C07278=1088.275,-115.195,449.756,174.378,16.605,152.666
C07279=1088.269,-115.445,449.766,174.377,16.605,152.667
C07280=1088.263,-115.695,449.776,174.375,16.604,152.667
C07281=1088.257,-115.945,449.785,174.373,16.603,152.667
C07282=1088.251,-116.194,449.795,174.372,16.603,152.667
C07283=1088.245,-116.444,449.804,174.370,16.603,152.667
C07284=1088.239,-116.693,449.813,174.369,16.602,152.668
C07285=1088.233,-116.943,449.823,174.368,16.602,152.668
C07286=1088.227,-117.193,449.833,174.366,16.601,152.668
C07287=1088.220,-117.443,449.842,174.364,16.600,152.668
C07288=1088.215,-117.693,449.851,174.363,16.600,152.668
C07289=1088.208,-117.943,449.861,174.361,16.599,152.669
C07290=1088.202,-118.193,449.870,174.359,16.598,152.669
C07291=1088.197,-118.442,449.879,174.358,16.598,152.669
C07292=1088.190,-118.691,449.888,174.356,16.597,152.669
C07293=1088.184,-118.941,449.898,174.355,16.596,152.669
C07294=1088.177,-119.191,449.907,174.354,16.596,152.670
C07295=1088.171,-119.441,449.917,174.352,16.596,152.670
C07296=1088.165,-119.691,449.927,174.350,16.595,152.670
C07297=1088.159,-119.941,449.935,174.348,16.594,152.670
C07298=1088.153,-120.191,449.945,174.347,16.594,152.670
C07299=1088.147,-120.440,449.954,174.345,16.593,152.671
C07300=1088.141,-120.689,449.963,174.343,16.592,152.671
C07301=1088.134,-120.939,449.973,174.342,16.592,152.671
C07302=1088.128,-121.189,449.982,174.340,16.592,152.671
C07303=1088.122,-121.439,449.991,174.340,16.591,152.671
C07304=1088.116,-121.689,450.001,174.338,16.590,152.672
C07305=1088.110,-121.939,450.010,174.336,16.590,152.672
C07306=1088.104,-122.188,450.019,174.335,16.590,152.672
C07307=1088.098,-122.438,450.028,174.333,16.589,152.672
C07308=1088.091,-122.687,450.038,174.331,16.588,152.673
C07309=1088.086,-122.938,450.047,174.330,16.588,152.673
C07310=1088.079,-123.188,450.056,174.328,16.587,152.673
C07311=1088.074,-123.437,450.066,174.326,16.586,152.673
C07312=1088.068,-123.686,450.075,174.325,16.586,152.673
C07313=1088.061,-123.937,450.083,174.323,16.586,152.674
C07314=1088.055,-124.186,450.093,174.322,16.585,152.674
C07315=1088.049,-124.436,450.103,174.321,16.585,152.674
C07316=1088.042,-124.686,450.112,174.319,16.584,152.674
C07317=1088.037,-124.936,450.121,174.317,16.583,152.674
C07318=1088.030,-125.185,450.130,174.316,16.583,152.675
C07319=1088.024,-125.435,450.139,174.314,16.583,152.675
C07320=1088.018,-125.685,450.149,174.312,16.582,152.675
C07321=1088.012,-125.935,450.158,174.311,16.582,152.675
C07322=1088.006,-126.184,450.166,174.309,16.581,152.676
C07323=1088.000,-126.434,450.176,174.308,16.581,152.676
C07324=1087.993,-126.684,450.185,174.306,16.580,152.676
C07325=1087.987,-126.934,450.194,174.304,16.580,152.676
C07326=1087.981,-127.183,450.203,174.303,16.580,152.677
C07327=1087.974,-127.433,450.213,174.302,16.579,152.677
C07328=1087.969,-127.683,450.221,174.300,16.578,152.677
C07329=1087.962,-127.941,450.231,174.299,16.578,152.677
C07330=1087.957,-128.198,450.240,174.297,16.577,152.677
C07331=1087.958,-128.455,450.252,174.296,16.575,152.677
C07332=1087.965,-128.710,450.265,174.296,16.571,152.676
C07333=1087.560,-128.731,450.140,174.254,16.677,152.705
C07334=1087.553,-128.477,450.127,174.254,16.681,152.706
C07335=1087.552,-128.220,450.115,174.255,16.683,152.706
C07336=1087.558,-127.963,450.105,174.257,16.684,152.706
C07337=1087.564,-127.705,450.096,174.258,16.684,152.705
C07338=1087.571,-127.455,450.086,174.260,16.685,152.705
C07339=1087.576,-127.205,450.078,174.262,16.686,152.705
C07340=1087.582,-126.955,450.068,174.263,16.686,152.705
C07341=1087.589,-126.706,450.059,174.265,16.687,152.705
C07342=1087.595,-126.456,450.050,174.267,16.687,152.704
C07343=1087.601,-126.206,450.041,174.268,16.687,152.704
C07344=1087.607,-125.957,450.031,174.270,16.688,152.704
C07345=1087.614,-125.707,450.022,174.271,16.689,152.704
C07346=1087.619,-125.457,450.014,174.272,16.689,152.703
C07347=1087.626,-125.207,450.004,174.274,16.690,152.703
C07348=1087.632,-124.957,449.995,174.275,16.690,152.703
C07349=1087.639,-124.708,449.986,174.277,16.691,152.703
C07350=1087.644,-124.458,449.977,174.279,16.691,152.703
C07351=1087.650,-124.208,449.967,174.280,16.691,152.702
C07352=1087.656,-123.958,449.958,174.282,16.692,152.702
C07353=1087.663,-123.709,449.949,174.284,16.693,152.702
C07354=1087.669,-123.458,449.940,174.285,16.693,152.702
C07355=1087.675,-123.209,449.931,174.287,16.694,152.701
C07356=1087.681,-122.960,449.921,174.289,16.694,152.701
C07357=1087.687,-122.710,449.912,174.289,16.695,152.701
C07358=1087.693,-122.460,449.902,174.291,16.696,152.701
C07359=1087.700,-122.210,449.894,174.293,16.696,152.701
C07360=1087.706,-121.960,449.884,174.294,16.697,152.701
C07361=1087.711,-121.711,449.875,174.296,16.697,152.700
C07362=1087.718,-121.461,449.866,174.298,16.698,152.700
C07363=1087.724,-121.211,449.856,174.299,16.698,152.700
C07364=1087.730,-120.961,449.847,174.301,16.699,152.700
C07365=1087.736,-120.711,449.838,174.303,16.700,152.699
C07366=1087.743,-120.462,449.829,174.304,16.700,152.699
C07367=1087.748,-120.213,449.819,174.305,16.701,152.699
C07368=1087.754,-119.963,449.810,174.307,16.701,152.699
C07369=1087.761,-119.713,449.800,174.308,16.701,152.699
C07370=1087.767,-119.463,449.791,174.310,16.702,152.698
C07371=1087.773,-119.213,449.782,174.312,16.703,152.698
C07372=1087.779,-118.963,449.772,174.313,16.703,152.698
C07373=1087.785,-118.713,449.763,174.315,16.704,152.698
C07374=1087.792,-118.464,449.754,174.316,16.705,152.698
C07375=1087.798,-118.215,449.745,174.318,16.705,152.697
C07376=1087.804,-117.965,449.735,174.319,16.706,152.697
C07377=1087.810,-117.715,449.725,174.321,16.706,152.697
C07378=1087.816,-117.465,449.716,174.323,16.708,152.697
C07379=1087.822,-117.215,449.706,174.324,16.708,152.697
C07380=1087.828,-116.966,449.697,174.326,16.708,152.696
C07381=1087.835,-116.716,449.687,174.327,16.709,152.696
C07382=1087.840,-116.465,449.678,174.329,16.709,152.696
C07383=1087.847,-116.216,449.669,174.330,16.710,152.696
C07384=1087.852,-115.967,449.660,174.332,16.711,152.696
C07385=1087.858,-115.717,449.650,174.333,16.711,152.696
C07386=1087.864,-115.467,449.640,174.335,16.712,152.695
C07387=1087.871,-115.217,449.631,174.337,16.713,152.695
C07388=1087.877,-114.967,449.621,174.338,16.714,152.695
C07389=1087.883,-114.718,449.612,174.339,16.714,152.695
C07390=1087.889,-114.468,449.602,174.341,16.714,152.695
C07391=1087.895,-114.218,449.593,174.343,16.716,152.694
C07392=1087.902,-113.968,449.583,174.344,16.716,152.694
C07393=1087.908,-113.718,449.573,174.346,16.717,152.694
C07394=1087.915,-113.448,449.563,174.348,16.717,152.694
C07395=1087.921,-113.177,449.553,174.349,16.718,152.694
C07396=1087.928,-112.907,449.542,174.351,16.719,152.693
C07397=1087.934,-112.635,449.532,174.353,16.720,152.693
C07398=1087.940,-112.385,449.523,174.354,16.720,152.693
C07399=1087.947,-112.135,449.513,174.356,16.721,152.693
C07400=1087.953,-111.886,449.503,174.358,16.722,152.693
C07401=1087.959,-111.636,449.494,174.359,16.722,152.693
C07402=1087.964,-111.387,449.485,174.360,16.723,152.692
C07403=1087.971,-111.137,449.475,174.362,16.724,152.692
C07404=1087.977,-110.887,449.466,174.364,16.725,152.692
C07405=1087.983,-110.638,449.455,174.365,16.725,152.692
C07406=1087.989,-110.388,449.446,174.367,16.726,152.692
C07407=1087.995,-110.138,449.436,174.368,16.726,152.691
C07408=1088.001,-109.888,449.426,174.369,16.727,152.691
C07409=1088.007,-109.639,449.416,174.371,16.728,152.691
C07410=1088.013,-109.389,449.407,174.373,16.729,152.691
C07411=1088.020,-109.139,449.397,174.375,16.729,152.691
C07412=1088.026,-108.889,449.388,174.376,16.730,152.691
C07413=1088.032,-108.639,449.378,174.377,16.730,152.690
C07414=1088.038,-108.390,449.369,174.379,16.731,152.690
C07415=1088.045,-108.140,449.358,174.381,16.732,152.690
C07416=1088.051,-107.891,449.349,174.382,16.733,152.690
C07417=1088.057,-107.641,449.339,174.383,16.734,152.690
C07418=1088.062,-107.391,449.329,174.385,16.734,152.690
C07419=1088.068,-107.141,449.319,174.387,16.735,152.689
C07420=1088.075,-106.891,449.310,174.388,16.735,152.689
C07421=1088.081,-106.642,449.300,174.390,16.737,152.689
C07422=1088.087,-106.392,449.290,174.392,16.737,152.689
C07423=1088.093,-106.142,449.280,174.393,16.738,152.689
C07424=1088.099,-105.892,449.270,174.394,16.739,152.689
C07425=1088.105,-105.642,449.261,174.396,16.739,152.688
C07426=1088.111,-105.393,449.251,174.398,16.740,152.688
C07427=1088.118,-105.143,449.241,174.400,16.741,152.688
C07428=1088.123,-104.893,449.231,174.400,16.742,152.688
C07429=1088.129,-104.643,449.221,174.402,16.743,152.688
C07430=1088.136,-104.394,449.212,174.404,16.743,152.688
C07431=1088.142,-104.145,449.201,174.406,16.744,152.687
C07432=1088.147,-103.894,449.191,174.407,16.746,152.687
C07433=1088.154,-103.645,449.182,174.408,16.746,152.687
C07434=1088.160,-103.395,449.172,174.410,16.747,152.687
C07435=1088.166,-103.145,449.162,174.412,16.747,152.687
C07436=1088.172,-102.896,449.152,174.413,16.748,152.687
C07437=1088.178,-102.646,449.142,174.414,16.749,152.687
C07438=1088.184,-102.396,449.132,174.416,16.750,152.686
C07439=1088.190,-102.147,449.122,174.418,16.751,152.686
C07440=1088.196,-101.897,449.112,174.419,16.752,152.686
C07441=1088.202,-101.647,449.102,174.421,16.752,152.686
C07442=1088.208,-101.397,449.093,174.422,16.753,152.686
C07443=1088.215,-101.148,449.083,174.424,16.754,152.686
C07444=1088.220,-100.898,449.072,174.426,16.755,152.685
C07445=1088.226,-100.648,449.063,174.427,16.756,152.685
C07446=1088.233,-100.399,449.053,174.428,16.756,152.685
C07447=1088.238,-100.149,449.042,174.430,16.757,152.685
C07448=1088.244,-99.899,449.033,174.432,16.758,152.685
C07449=1088.251,-99.650,449.023,174.433,16.759,152.685
C07450=1088.257,-99.400,449.013,174.435,16.760,152.684
C07451=1088.263,-99.150,449.003,174.436,16.760,152.684
C07452=1088.269,-98.901,448.992,174.438,16.761,152.684
C07453=1088.275,-98.651,448.983,174.440,16.762,152.684
C07454=1088.281,-98.401,448.973,174.441,16.763,152.684
C07455=1088.288,-98.151,448.962,174.443,16.764,152.684
C07456=1088.294,-97.901,448.953,174.444,16.765,152.684
C07457=1088.300,-97.652,448.942,174.446,16.765,152.684
C07458=1088.306,-97.375,448.931,174.447,16.766,152.683
C07459=1088.312,-97.099,448.920,174.449,16.767,152.683
C07460=1088.319,-96.822,448.909,174.451,16.769,152.683
C07461=1088.326,-96.546,448.897,174.452,16.769,152.683
C07462=1088.331,-96.296,448.887,174.454,16.770,152.683
C07463=1088.338,-96.047,448.877,174.456,16.771,152.683
C07464=1088.343,-95.796,448.867,174.457,16.772,152.683
C07465=1088.349,-95.547,448.857,174.458,16.773,152.683
C07466=1088.356,-95.296,448.846,174.460,16.774,152.682
C07467=1088.362,-95.047,448.836,174.462,16.775,152.682
C07468=1088.368,-94.797,448.826,174.463,16.776,152.682
C07469=1088.374,-94.547,448.816,174.465,16.777,152.682
C07470=1088.380,-94.298,448.806,174.467,16.778,152.682
C07471=1088.386,-94.048,448.795,174.468,16.778,152.682
C07472=1088.392,-93.799,448.785,174.469,16.779,152.681
C07473=1088.398,-93.549,448.775,174.471,16.780,152.681
C07474=1088.403,-93.299,448.765,174.473,16.781,152.681
C07475=1088.410,-93.050,448.755,174.474,16.782,152.681
C07476=1088.415,-92.799,448.744,174.476,16.784,152.681
C07477=1088.422,-92.550,448.734,174.477,16.784,152.681
C07478=1088.427,-92.300,448.724,174.479,16.785,152.681
C07479=1088.434,-92.050,448.713,174.480,16.786,152.681
C07480=1088.440,-91.801,448.702,174.482,16.787,152.680
C07481=1088.446,-91.551,448.693,174.484,16.788,152.680
C07482=1088.452,-91.301,448.682,174.485,16.789,152.680
C07483=1088.458,-91.052,448.672,174.486,16.789,152.680
C07484=1088.464,-90.802,448.662,174.488,16.790,152.680
C07485=1088.470,-90.552,448.652,174.490,16.791,152.680
C07486=1088.475,-90.303,448.641,174.491,16.792,152.680
C07487=1088.482,-90.053,448.632,174.493,16.794,152.680
C07488=1088.488,-89.803,448.620,174.494,16.795,152.679
C07489=1088.494,-89.553,448.609,174.495,16.795,152.679
C07490=1088.500,-89.304,448.600,174.497,16.796,152.679
C07491=1088.506,-89.054,448.589,174.499,16.797,152.679
C07492=1088.512,-88.804,448.579,174.500,16.798,152.679
C07493=1088.518,-88.555,448.569,174.502,16.799,152.679
C07494=1088.524,-88.306,448.558,174.504,16.800,152.679
C07495=1088.530,-88.055,448.548,174.505,16.801,152.679
C07496=1088.537,-87.806,448.537,174.506,16.802,152.679
C07497=1088.542,-87.556,448.527,174.508,16.803,152.678
C07498=1088.548,-87.306,448.516,174.509,16.804,152.678
C07499=1088.554,-87.057,448.506,174.511,16.805,152.678
C07500=1088.560,-86.806,448.496,174.513,16.806,152.678
C07501=1088.567,-86.557,448.485,174.515,16.807,152.678
C07502=1088.572,-86.307,448.474,174.516,16.808,152.678
C07503=1088.578,-86.057,448.464,174.517,16.809,152.678
C07504=1088.584,-85.808,448.454,174.519,16.810,152.678
C07505=1088.590,-85.559,448.443,174.520,16.811,152.677
C07506=1088.597,-85.308,448.433,174.522,16.812,152.677
C07507=1088.603,-85.059,448.422,174.524,16.813,152.677
C07508=1088.608,-84.809,448.411,174.525,16.814,152.677
C07509=1088.615,-84.560,448.401,174.527,16.815,152.677
C07510=1088.621,-84.309,448.391,174.529,16.816,152.677
C07511=1088.627,-84.060,448.380,174.530,16.816,152.677
C07512=1088.633,-83.810,448.369,174.531,16.817,152.677
C07513=1088.639,-83.560,448.359,174.533,16.819,152.676
C07514=1088.645,-83.311,448.349,174.534,16.820,152.676
C07515=1088.651,-83.061,448.338,174.536,16.821,152.676
C07516=1088.657,-82.812,448.327,174.538,16.822,152.676
C07517=1088.663,-82.562,448.317,174.539,16.823,152.676
C07518=1088.669,-82.312,448.306,174.541,16.824,152.676
C07519=1088.676,-82.062,448.296,174.542,16.825,152.676
C07520=1088.682,-81.813,448.285,174.543,16.826,152.676
C07521=1088.688,-81.563,448.274,174.545,16.827,152.676
C07522=1088.695,-81.289,448.263,174.547,16.828,152.676
C07523=1088.701,-81.015,448.251,174.548,16.829,152.675
C07524=1088.707,-80.740,448.239,174.551,16.831,152.675
C07525=1088.715,-80.466,448.228,174.553,16.831,152.675
C07526=1088.721,-80.216,448.217,174.553,16.832,152.675
C07527=1088.727,-79.966,448.207,174.555,16.833,152.675
C07528=1088.733,-79.717,448.196,174.557,16.834,152.675
C07529=1088.739,-79.467,448.185,174.558,16.835,152.675
C07530=1088.745,-79.217,448.174,174.560,16.836,152.675
C07531=1088.751,-78.968,448.163,174.561,16.838,152.675
C07532=1088.756,-78.718,448.152,174.563,16.839,152.674
C07533=1088.763,-78.468,448.143,174.565,16.840,152.674
C07534=1088.769,-78.218,448.131,174.566,16.841,152.674
C07535=1088.775,-77.969,448.121,174.568,16.842,152.674
C07536=1088.780,-77.719,448.110,174.570,16.843,152.674
C07537=1088.786,-77.470,448.099,174.570,16.844,152.674
C07538=1088.793,-77.220,448.088,174.572,16.845,152.674
C07539=1088.799,-76.970,448.077,174.574,16.846,152.674
C07540=1088.805,-76.721,448.066,174.575,16.847,152.674
C07541=1088.810,-76.471,448.055,174.577,16.848,152.674
C07542=1088.816,-76.220,448.045,174.578,16.850,152.673
C07543=1088.822,-75.971,448.034,174.580,16.851,152.673
C07544=1088.828,-75.722,448.023,174.582,16.852,152.673
C07545=1088.835,-75.472,448.013,174.583,16.853,152.673
C07546=1088.841,-75.222,448.002,174.585,16.854,152.673
C07547=1088.846,-74.973,447.991,174.587,16.855,152.673
C07548=1088.852,-74.723,447.980,174.588,16.856,152.673
C07549=1088.859,-74.473,447.969,174.590,16.858,152.673
C07550=1088.864,-74.223,447.958,174.591,16.859,152.673
C07551=1088.870,-73.974,447.947,174.592,16.859,152.673
C07552=1088.876,-73.724,447.936,174.594,16.861,152.673
C07553=1088.882,-73.474,447.925,174.595,16.862,152.672
C07554=1088.888,-73.225,447.914,174.597,16.863,152.672
C07555=1088.894,-72.975,447.903,174.599,16.864,152.672
C07556=1088.900,-72.725,447.892,174.600,16.865,152.672
C07557=1088.906,-72.476,447.881,174.602,16.867,152.672
C07558=1088.911,-72.226,447.870,174.603,16.868,152.672
C07559=1088.917,-71.977,447.859,174.605,16.869,152.672
C07560=1088.923,-71.726,447.848,174.606,16.870,152.672
C07561=1088.929,-71.477,447.837,174.608,16.871,152.672
C07562=1088.935,-71.228,447.826,174.609,16.873,152.672
C07563=1088.941,-70.978,447.815,174.611,16.874,152.672
C07564=1088.947,-70.728,447.804,174.613,16.875,152.672
C07565=1088.953,-70.478,447.793,174.614,16.876,152.671
C07566=1088.958,-70.229,447.782,174.616,16.877,152.671
C07567=1088.964,-69.978,447.770,174.617,16.879,152.671
C07568=1088.970,-69.729,447.760,174.619,16.880,152.671
C07569=1088.976,-69.479,447.749,174.621,16.881,152.671
C07570=1088.982,-69.230,447.737,174.622,16.882,152.671
C07571=1088.988,-68.980,447.726,174.623,16.883,152.671
C07572=1088.994,-68.731,447.715,174.624,16.884,152.671
C07573=1088.999,-68.481,447.704,174.626,16.885,152.671
C07574=1089.006,-68.231,447.693,174.628,16.886,152.671
C07575=1089.012,-67.982,447.682,174.629,16.887,152.671
C07576=1089.017,-67.732,447.671,174.631,16.889,152.671
C07577=1089.023,-67.482,447.659,174.632,16.890,152.671
C07578=1089.029,-67.232,447.648,174.634,16.891,152.671
C07579=1089.035,-66.983,447.636,174.636,16.892,152.670
C07580=1089.041,-66.733,447.626,174.637,16.893,152.670
C07581=1089.047,-66.484,447.615,174.639,16.895,152.670
C07582=1089.053,-66.233,447.603,174.640,16.896,152.670
C07583=1089.059,-65.984,447.593,174.642,16.897,152.670
C07584=1089.065,-65.734,447.582,174.643,16.898,152.670
C07585=1089.071,-65.485,447.570,174.645,16.900,152.670
C07586=1089.077,-65.213,447.557,174.646,16.901,152.670
C07587=1089.084,-64.941,447.545,174.648,16.902,152.670
C07588=1089.090,-64.668,447.533,174.650,16.904,152.670
C07589=1089.097,-64.396,447.521,174.652,16.905,152.670
C07590=1089.102,-64.147,447.510,174.654,16.906,152.669
C07591=1089.109,-63.897,447.499,174.655,16.908,152.670
C07592=1089.114,-63.647,447.487,174.657,16.909,152.669
C07593=1089.120,-63.398,447.475,174.658,16.910,152.669
C07594=1089.126,-63.148,447.464,174.660,16.911,152.669
C07595=1089.132,-62.898,447.453,174.661,16.913,152.669
C07596=1089.138,-62.648,447.442,174.663,16.914,152.669
C07597=1089.144,-62.399,447.430,174.665,16.915,152.669
C07598=1089.150,-62.149,447.419,174.666,16.916,152.669
C07599=1089.156,-61.899,447.408,174.668,16.918,152.669
C07600=1089.162,-61.650,447.396,174.669,16.919,152.669
C07601=1089.168,-61.400,447.385,174.671,16.920,152.669
C07602=1089.174,-61.151,447.374,174.672,16.921,152.669
C07603=1089.180,-60.901,447.362,174.674,16.922,152.669
C07604=1089.185,-60.651,447.351,174.675,16.924,152.669
C07605=1089.192,-60.401,447.339,174.677,16.925,152.668
C07606=1089.198,-60.152,447.328,174.679,16.926,152.668
C07607=1089.204,-59.902,447.317,174.680,16.927,152.668
C07608=1089.210,-59.653,447.306,174.682,16.929,152.668
C07609=1089.215,-59.403,447.293,174.683,16.930,152.668
C07610=1089.222,-59.153,447.282,174.685,16.931,152.668
C07611=1089.227,-58.904,447.271,174.686,16.932,152.668
C07612=1089.234,-58.654,447.259,174.688,16.933,152.668
C07613=1089.239,-58.404,447.248,174.690,16.935,152.668
C07614=1089.245,-58.154,447.237,174.691,16.936,152.668
C07615=1089.251,-57.905,447.225,174.693,16.937,152.668
C07616=1089.258,-57.655,447.214,174.694,16.938,152.668
C07617=1089.264,-57.406,447.202,174.696,16.939,152.668
C07618=1089.269,-57.156,447.190,174.697,16.941,152.668
C07619=1089.275,-56.907,447.179,174.699,16.942,152.668
C07620=1089.282,-56.657,447.168,174.700,16.943,152.667
C07621=1089.287,-56.407,447.157,174.702,16.944,152.667
C07622=1089.293,-56.157,447.144,174.704,16.946,152.667
C07623=1089.300,-55.907,447.133,174.705,16.947,152.667
C07624=1089.306,-55.658,447.121,174.707,16.948,152.667
C07625=1089.312,-55.408,447.110,174.708,16.949,152.667
C07626=1089.317,-55.159,447.098,174.710,16.951,152.667
C07627=1089.324,-54.909,447.087,174.711,16.952,152.667
C07628=1089.330,-54.660,447.075,174.713,16.953,152.667
C07629=1089.336,-54.410,447.064,174.715,16.954,152.667
C07630=1089.341,-54.161,447.052,174.716,16.956,152.667
C07631=1089.348,-53.910,447.040,174.718,16.957,152.667
C07632=1089.354,-53.661,447.028,174.719,16.958,152.667
C07633=1089.360,-53.411,447.018,174.721,16.959,152.667
C07634=1089.366,-53.161,447.005,174.722,16.961,152.667
C07635=1089.372,-52.912,446.994,174.724,16.962,152.666
C07636=1089.378,-52.662,446.982,174.725,16.963,152.666
C07637=1089.383,-52.412,446.971,174.727,16.965,152.666
C07638=1089.390,-52.163,446.959,174.728,16.966,152.666
C07639=1089.396,-51.913,446.947,174.730,16.967,152.666
C07640=1089.402,-51.664,446.935,174.732,16.968,152.666
C07641=1089.408,-51.414,446.923,174.734,16.970,152.666
C07642=1089.414,-51.164,446.912,174.735,16.971,152.666
C07643=1089.421,-50.915,446.900,174.737,16.972,152.666
C07644=1089.426,-50.664,446.889,174.738,16.974,152.666
C07645=1089.432,-50.416,446.877,174.740,16.975,152.666
C07646=1089.438,-50.166,446.865,174.742,16.976,152.666
C07647=1089.444,-49.916,446.854,174.743,16.978,152.666
C07648=1089.450,-49.666,446.841,174.745,16.979,152.666
C07649=1089.456,-49.417,446.830,174.746,16.980,152.666
C07650=1089.462,-49.146,446.816,174.748,16.982,152.666
C07651=1089.469,-48.875,446.804,174.749,16.983,152.666
C07652=1089.474,-48.604,446.791,174.751,16.985,152.666
C07653=1089.481,-48.334,446.779,174.753,16.986,152.665
C07654=1089.487,-48.084,446.766,174.754,16.988,152.665
C07655=1089.494,-47.834,446.754,174.756,16.989,152.665
C07656=1089.499,-47.584,446.743,174.758,16.990,152.665
C07657=1089.505,-47.335,446.731,174.759,16.991,152.665
C07658=1089.510,-47.086,446.718,174.761,16.992,152.665
C07659=1089.517,-46.835,446.707,174.762,16.994,152.665
C07660=1089.522,-46.586,446.695,174.764,16.995,152.665
C07661=1089.529,-46.337,446.683,174.765,16.996,152.665
C07662=1089.534,-46.086,446.671,174.768,16.998,152.665
C07663=1089.540,-45.837,446.659,174.769,17.000,152.665
C07664=1089.546,-45.587,446.647,174.770,17.001,152.665
C07665=1089.552,-45.338,446.635,174.772,17.002,152.665
C07666=1089.558,-45.088,446.624,174.774,17.003,152.665
C07667=1089.564,-44.838,446.611,174.775,17.005,152.665
C07668=1089.569,-44.589,446.599,174.777,17.006,152.665
C07669=1089.576,-44.339,446.587,174.778,17.008,152.665
C07670=1089.581,-44.089,446.575,174.780,17.009,152.665
C07671=1089.587,-43.840,446.564,174.781,17.010,152.665
C07672=1089.593,-43.590,446.551,174.783,17.012,152.665
C07673=1089.599,-43.341,446.539,174.784,17.013,152.664
C07674=1089.605,-43.091,446.527,174.786,17.014,152.665
C07675=1089.611,-42.841,446.515,174.788,17.016,152.664
C07676=1089.617,-42.592,446.503,174.789,17.018,152.664
C07677=1089.623,-42.342,446.491,174.791,17.019,152.664
C07678=1089.629,-42.092,446.478,174.793,17.020,152.664
C07679=1089.635,-41.843,446.467,174.794,17.021,152.664
C07680=1089.640,-41.593,446.455,174.796,17.022,152.664
C07681=1089.646,-41.343,446.442,174.797,17.024,152.664
C07682=1089.652,-41.094,446.431,174.799,17.025,152.664
C07683=1089.658,-40.844,446.418,174.800,17.026,152.664
C07684=1089.665,-40.595,446.406,174.802,17.028,152.664
C07685=1089.670,-40.345,446.394,174.803,17.029,152.664
C07686=1089.676,-40.096,446.381,174.806,17.031,152.664
C07687=1089.683,-39.845,446.370,174.807,17.032,152.664
C07688=1089.688,-39.596,446.358,174.809,17.034,152.664
C07689=1089.694,-39.346,446.345,174.810,17.035,152.664
C07690=1089.700,-39.097,446.334,174.812,17.036,152.664
C07691=1089.706,-38.847,446.321,174.813,17.038,152.664
C07692=1089.712,-38.598,446.309,174.815,17.039,152.664
C07693=1089.717,-38.348,446.296,174.816,17.040,152.664
C07694=1089.724,-38.098,446.284,174.818,17.042,152.664
C07695=1089.729,-37.849,446.272,174.820,17.044,152.664
C07696=1089.735,-37.599,446.260,174.822,17.045,152.663
C07697=1089.741,-37.349,446.247,174.823,17.046,152.663
C07698=1089.747,-37.100,446.235,174.825,17.048,152.663
C07699=1089.753,-36.851,446.223,174.826,17.049,152.663
C07700=1089.759,-36.601,446.210,174.828,17.050,152.663
C07701=1089.764,-36.351,446.198,174.829,17.052,152.663
C07702=1089.770,-36.102,446.186,174.831,17.053,152.663
C07703=1089.776,-35.852,446.173,174.832,17.055,152.663
C07704=1089.781,-35.602,446.162,174.834,17.056,152.663
C07705=1089.788,-35.352,446.150,174.836,17.058,152.663
C07706=1089.794,-35.103,446.136,174.837,17.059,152.663
C07707=1089.800,-34.853,446.124,174.839,17.061,152.663
C07708=1089.805,-34.604,446.112,174.840,17.062,152.663
C07709=1089.811,-34.354,446.099,174.842,17.063,152.663
C07710=1089.817,-34.104,446.086,174.843,17.064,152.663
C07711=1089.823,-33.854,446.074,174.845,17.066,152.663
C07712=1089.829,-33.606,446.062,174.847,17.068,152.663
C07713=1089.835,-33.356,446.050,174.848,17.069,152.663
C07714=1089.841,-33.085,446.036,174.850,17.070,152.663
C07715=1089.847,-32.815,446.022,174.851,17.072,152.663
C07716=1089.854,-32.544,446.009,174.854,17.074,152.663
C07717=1089.860,-32.273,445.996,174.855,17.075,152.663
C07718=1089.866,-32.024,445.983,174.857,17.076,152.663
C07719=1089.872,-31.774,445.970,174.858,17.078,152.663
C07720=1089.878,-31.525,445.958,174.860,17.079,152.663
C07721=1089.883,-31.275,445.946,174.862,17.081,152.663
C07722=1089.889,-31.025,445.933,174.864,17.082,152.663
C07723=1089.895,-30.775,445.920,174.865,17.084,152.663
C07724=1089.901,-30.527,445.909,174.867,17.085,152.662
C07725=1089.907,-30.277,445.896,174.868,17.087,152.663
C07726=1089.913,-30.027,445.883,174.870,17.088,152.662
C07727=1089.919,-29.778,445.871,174.871,17.089,152.662
C07728=1089.925,-29.528,445.858,174.873,17.091,152.662
C07729=1089.931,-29.278,445.846,174.875,17.092,152.662
C07730=1089.937,-29.029,445.833,174.876,17.094,152.662
C07731=1089.943,-28.779,445.820,174.878,17.095,152.662
C07732=1089.949,-28.529,445.807,174.879,17.096,152.662
C07733=1089.955,-28.280,445.795,174.881,17.098,152.662
C07734=1089.960,-28.030,445.782,174.882,17.099,152.662
C07735=1089.966,-27.780,445.770,174.885,17.101,152.662
C07736=1089.972,-27.531,445.757,174.886,17.102,152.662
C07737=1089.979,-27.282,445.745,174.888,17.103,152.662
C07738=1089.985,-27.032,445.732,174.889,17.105,152.662
C07739=1089.990,-26.782,445.720,174.891,17.106,152.662
C07740=1089.996,-26.532,445.706,174.892,17.108,152.662
C07741=1090.001,-26.283,445.694,174.894,17.109,152.662
C07742=1090.007,-26.033,445.681,174.896,17.111,152.662
C07743=1090.013,-25.783,445.669,174.898,17.112,152.662
C07744=1090.019,-25.534,445.655,174.899,17.114,152.662
C07745=1090.025,-25.284,445.643,174.900,17.115,152.662
C07746=1090.030,-25.035,445.631,174.902,17.116,152.662
C07747=1090.037,-24.786,445.617,174.903,17.118,152.662
C07748=1090.043,-24.536,445.605,174.906,17.120,152.662
C07749=1090.048,-24.286,445.592,174.907,17.121,152.662
C07750=1090.054,-24.036,445.579,174.909,17.122,152.662
C07751=1090.060,-23.787,445.566,174.910,17.124,152.662
C07752=1090.065,-23.537,445.554,174.912,17.125,152.662
C07753=1090.071,-23.287,445.541,174.914,17.127,152.662
C07754=1090.077,-23.038,445.528,174.915,17.129,152.662
C07755=1090.083,-22.788,445.515,174.917,17.130,152.661
C07756=1090.089,-22.539,445.502,174.918,17.132,152.662
C07757=1090.095,-22.289,445.489,174.920,17.133,152.661
C07758=1090.100,-22.039,445.476,174.921,17.134,152.661
C07759=1090.106,-21.790,445.463,174.924,17.136,152.661
C07760=1090.112,-21.541,445.451,174.925,17.138,152.661
C07761=1090.118,-21.291,445.438,174.927,17.139,152.661
C07762=1090.124,-21.041,445.425,174.928,17.140,152.661
C07763=1090.129,-20.791,445.412,174.930,17.141,152.661
C07764=1090.136,-20.542,445.399,174.931,17.143,152.661
C07765=1090.141,-20.292,445.386,174.933,17.145,152.661
C07766=1090.148,-20.043,445.373,174.935,17.146,152.661
C07767=1090.154,-19.793,445.360,174.936,17.147,152.661
C07768=1090.158,-19.544,445.347,174.938,17.149,152.661
C07769=1090.164,-19.294,445.334,174.939,17.151,152.661
C07770=1090.170,-19.044,445.322,174.942,17.152,152.661
C07771=1090.176,-18.795,445.308,174.943,17.154,152.661
C07772=1090.182,-18.545,445.296,174.945,17.155,152.661
C07773=1090.189,-18.296,445.282,174.946,17.157,152.661
C07774=1090.194,-18.046,445.269,174.948,17.158,152.661
C07775=1090.200,-17.796,445.256,174.950,17.160,152.661
C07776=1090.206,-17.546,445.244,174.951,17.161,152.661
C07777=1090.212,-17.297,445.230,174.953,17.163,152.661
C07778=1090.218,-17.026,445.216,174.954,17.164,152.661
C07779=1090.225,-16.755,445.202,174.957,17.166,152.661
C07780=1090.231,-16.484,445.188,174.958,17.167,152.661
C07781=1090.237,-16.213,445.173,174.960,17.169,152.661
C07782=1090.243,-15.963,445.160,174.962,17.170,152.661
C07783=1090.249,-15.713,445.147,174.963,17.172,152.661
C07784=1090.255,-15.464,445.135,174.965,17.173,152.661
C07785=1090.261,-15.214,445.121,174.966,17.175,152.661
C07786=1090.267,-14.964,445.108,174.968,17.176,152.661
C07787=1090.273,-14.715,445.095,174.970,17.178,152.660
C07788=1090.278,-14.465,445.081,174.972,17.179,152.661
C07789=1090.284,-14.215,445.069,174.973,17.181,152.660
C07790=1090.290,-13.966,445.055,174.975,17.182,152.660
C07791=1090.296,-13.716,445.041,174.977,17.184,152.660
C07792=1090.302,-13.467,445.029,174.978,17.185,152.660
C07793=1090.307,-13.217,445.015,174.980,17.187,152.660
C07794=1090.313,-12.967,445.002,174.981,17.188,152.660
C07795=1090.319,-12.718,444.989,174.983,17.190,152.660
C07796=1090.325,-12.468,444.975,174.985,17.191,152.660
C07797=1090.331,-12.218,444.963,174.986,17.193,152.660
C07798=1090.336,-11.969,444.949,174.988,17.194,152.660
C07799=1090.342,-11.720,444.936,174.989,17.196,152.660
C07800=1090.348,-11.469,444.922,174.991,17.197,152.660
C07801=1090.354,-11.220,444.909,174.993,17.199,152.660
C07802=1090.359,-10.971,444.895,174.995,17.201,152.660
C07803=1090.365,-10.721,444.882,174.996,17.202,152.660
C07804=1090.371,-10.471,444.870,174.998,17.203,152.660
C07805=1090.377,-10.222,444.856,175.000,17.205,152.660
C07806=1090.383,-9.973,444.842,175.001,17.207,152.660
C07807=1090.388,-9.722,444.829,175.003,17.208,152.660
C07808=1090.394,-9.473,444.816,175.004,17.209,152.660
C07809=1090.400,-9.224,444.802,175.006,17.211,152.660
C07810=1090.406,-8.974,444.789,175.008,17.212,152.660
C07811=1090.411,-8.724,444.776,175.010,17.214,152.660
C07812=1090.418,-8.475,444.762,175.011,17.215,152.660
C07813=1090.423,-8.225,444.749,175.013,17.217,152.660
C07814=1090.429,-7.976,444.735,175.015,17.218,152.660
C07815=1090.435,-7.727,444.722,175.016,17.220,152.660
C07816=1090.441,-7.477,444.709,175.018,17.221,152.660
C07817=1090.447,-7.227,444.696,175.019,17.223,152.660
C07818=1090.452,-6.978,444.682,175.022,17.224,152.660
C07819=1090.459,-6.728,444.668,175.023,17.226,152.660
C07820=1090.464,-6.479,444.655,175.025,17.228,152.660
C07821=1090.470,-6.230,444.641,175.026,17.229,152.660
C07822=1090.476,-5.979,444.628,175.028,17.230,152.660
C07823=1090.482,-5.729,444.615,175.030,17.232,152.659
C07824=1090.488,-5.480,444.601,175.031,17.234,152.660
C07825=1090.494,-5.231,444.587,175.033,17.235,152.659
C07826=1090.499,-4.981,444.574,175.034,17.236,152.660
C07827=1090.506,-4.732,444.560,175.037,17.238,152.659
C07828=1090.511,-4.482,444.546,175.038,17.240,152.659
C07829=1090.517,-4.233,444.533,175.040,17.241,152.659
C07830=1090.523,-3.983,444.519,175.041,17.242,152.659
C07831=1090.529,-3.733,444.506,175.044,17.244,152.659
C07832=1090.535,-3.483,444.492,175.045,17.246,152.659
C07833=1090.540,-3.234,444.479,175.047,17.247,152.659
C07834=1090.546,-2.984,444.465,175.048,17.248,152.659
C07835=1090.552,-2.735,444.451,175.050,17.250,152.659
C07836=1090.557,-2.485,444.438,175.052,17.251,152.659
C07837=1090.563,-2.236,444.424,175.053,17.253,152.659
C07838=1090.569,-1.986,444.410,175.055,17.254,152.659
C07839=1090.575,-1.737,444.397,175.057,17.256,152.659
C07840=1090.580,-1.487,444.383,175.059,17.257,152.659
C07841=1090.586,-1.238,444.369,175.060,17.259,152.659
C07842=1090.592,-0.964,444.354,175.062,17.261,152.659
C07843=1090.599,-0.692,444.339,175.064,17.262,152.659
C07844=1090.605,-0.418,444.324,175.066,17.264,152.659
C07845=1090.611,-0.146,444.309,175.067,17.266,152.659
C07846=1090.617,0.103,444.295,175.069,17.267,152.659
C07847=1090.623,0.353,444.281,175.071,17.269,152.659
C07848=1090.628,0.603,444.267,175.073,17.270,152.659
C07849=1090.635,0.852,444.254,175.074,17.272,152.659
C07850=1090.640,1.102,444.240,175.076,17.273,152.659
C07851=1090.645,1.351,444.226,175.078,17.275,152.659
C07852=1090.651,1.601,444.212,175.079,17.277,152.659
C07853=1090.656,1.851,444.198,175.081,17.278,152.659
C07854=1090.663,2.100,444.185,175.082,17.280,152.659
C07855=1090.669,2.350,444.171,175.085,17.281,152.659
C07856=1090.674,2.600,444.157,175.086,17.283,152.659
C07857=1090.680,2.849,444.143,175.088,17.284,152.659
C07858=1090.685,3.098,444.129,175.090,17.286,152.659
C07859=1090.692,3.347,444.115,175.092,17.287,152.658
C07860=1090.697,3.597,444.102,175.093,17.289,152.659
C07861=1090.703,3.847,444.087,175.094,17.290,152.659
C07862=1090.709,4.097,444.073,175.097,17.292,152.658
C07863=1090.714,4.346,444.060,175.098,17.294,152.658
C07864=1090.721,4.595,444.046,175.100,17.295,152.658
C07865=1090.726,4.845,444.032,175.101,17.296,152.658
C07866=1090.732,5.094,444.018,175.104,17.298,152.658
C07867=1090.738,5.345,444.004,175.105,17.300,152.658
C07868=1090.743,5.594,443.990,175.107,17.301,152.658
C07869=1090.749,5.844,443.976,175.109,17.303,152.658
C07870=1090.755,6.092,443.962,175.110,17.304,152.658
C07871=1090.761,6.343,443.948,175.112,17.306,152.658
C07872=1090.767,6.592,443.934,175.113,17.307,152.658
C07873=1090.772,6.842,443.920,175.116,17.309,152.658
C07874=1090.778,7.091,443.905,175.117,17.310,152.658
C07875=1090.783,7.340,443.892,175.119,17.312,152.658
C07876=1090.790,7.590,443.878,175.121,17.313,152.658
C07877=1090.796,7.840,443.864,175.122,17.315,152.658
C07878=1090.802,8.089,443.849,175.124,17.316,152.658
C07879=1090.807,8.338,443.836,175.125,17.318,152.658
C07880=1090.813,8.589,443.821,175.128,17.319,152.658
C07881=1090.819,8.838,443.807,175.129,17.321,152.658
C07882=1090.824,9.087,443.793,175.131,17.322,152.658
C07883=1090.830,9.337,443.779,175.133,17.324,152.658
C07884=1090.837,9.587,443.765,175.135,17.325,152.658
C07885=1090.842,9.836,443.751,175.136,17.327,152.658
C07886=1090.848,10.085,443.737,175.138,17.328,152.658
C07887=1090.854,10.335,443.722,175.140,17.330,152.658
C07888=1090.860,10.584,443.708,175.141,17.331,152.658
C07889=1090.865,10.834,443.694,175.143,17.333,152.658
C07890=1090.872,11.084,443.679,175.145,17.334,152.657
C07891=1090.877,11.333,443.665,175.147,17.336,152.657
C07892=1090.883,11.583,443.652,175.148,17.337,152.657
C07893=1090.889,11.833,443.637,175.150,17.339,152.657
C07894=1090.894,12.082,443.623,175.152,17.340,152.657
C07895=1090.901,12.331,443.609,175.154,17.341,152.657
C07896=1090.907,12.581,443.595,175.155,17.343,152.657
C07897=1090.913,12.831,443.581,175.157,17.345,152.657
C07898=1090.918,13.080,443.566,175.159,17.346,152.657
C07899=1090.924,13.330,443.552,175.160,17.347,152.657
C07900=1090.930,13.579,443.537,175.163,17.350,152.657
C07901=1090.936,13.828,443.523,175.164,17.351,152.657
C07902=1090.942,14.078,443.508,175.166,17.352,152.657
C07903=1090.947,14.328,443.495,175.167,17.353,152.657
C07904=1090.953,14.577,443.480,175.170,17.355,152.657
C07905=1090.959,14.827,443.466,175.171,17.357,152.657
C07906=1090.965,15.102,443.450,175.174,17.358,152.657
C07907=1090.972,15.376,443.434,175.175,17.360,152.657
C07908=1090.977,15.651,443.419,175.177,17.362,152.657
C07909=1090.985,15.926,443.403,175.179,17.363,152.657
C07910=1090.991,16.175,443.388,175.181,17.365,152.657
C07911=1090.995,16.425,443.374,175.183,17.366,152.657
C07912=1091.002,16.675,443.359,175.184,17.367,152.656
C07913=1091.007,16.924,443.345,175.186,17.370,152.656
C07914=1091.013,17.173,443.330,175.188,17.371,152.656
C07915=1091.019,17.423,443.315,175.189,17.372,152.656
C07916=1091.025,17.673,443.301,175.192,17.374,152.656
C07917=1091.031,17.922,443.287,175.193,17.376,152.656
C07918=1091.037,18.172,443.273,175.195,17.377,152.656
C07919=1091.042,18.421,443.257,175.197,17.379,152.656
C07920=1091.048,18.671,443.243,175.199,17.380,152.656
C07921=1091.054,18.920,443.229,175.200,17.382,152.656
C07922=1091.059,19.169,443.214,175.202,17.383,152.656
C07923=1091.065,19.420,443.200,175.204,17.384,152.656
C07924=1091.071,19.669,443.185,175.205,17.386,152.656
C07925=1091.076,19.918,443.170,175.207,17.387,152.656
C07926=1091.082,20.168,443.156,175.209,17.389,152.656
C07927=1091.088,20.417,443.141,175.211,17.390,152.656
C07928=1091.094,20.667,443.126,175.212,17.392,152.656
C07929=1091.100,20.916,443.112,175.215,17.393,152.656
C07930=1091.105,21.166,443.097,175.216,17.395,152.656
C07931=1091.111,21.415,443.082,175.218,17.396,152.656
C07932=1091.117,21.665,443.068,175.220,17.398,152.656
C07933=1091.123,21.914,443.054,175.222,17.399,152.656
C07934=1091.128,22.164,443.038,175.223,17.401,152.656
C07935=1091.134,22.413,443.024,175.225,17.403,152.656
C07936=1091.140,22.663,443.010,175.227,17.404,152.655
C07937=1091.145,22.912,442.994,175.228,17.405,152.656
C07938=1091.152,23.162,442.979,175.231,17.407,152.655
C07939=1091.157,23.411,442.966,175.232,17.409,152.655
C07940=1091.163,23.661,442.951,175.235,17.410,152.655
C07941=1091.168,23.910,442.935,175.236,17.411,152.655
C07942=1091.174,24.159,442.921,175.238,17.413,152.655
C07943=1091.180,24.410,442.907,175.240,17.415,152.655
C07944=1091.185,24.659,442.891,175.241,17.416,152.655
C07945=1091.192,24.909,442.877,175.243,17.417,152.655
C07946=1091.197,25.158,442.862,175.246,17.419,152.655
C07947=1091.203,25.407,442.846,175.247,17.421,152.655
C07948=1091.209,25.657,442.833,175.249,17.422,152.655
C07949=1091.215,25.907,442.818,175.251,17.424,152.655
C07950=1091.220,26.156,442.802,175.252,17.425,152.655
C07951=1091.226,26.406,442.787,175.254,17.426,152.655
C07952=1091.232,26.655,442.773,175.256,17.428,152.655
C07953=1091.238,26.905,442.757,175.258,17.429,152.655
C07954=1091.243,27.154,442.743,175.259,17.430,152.654
C07955=1091.250,27.404,442.729,175.262,17.433,152.655
C07956=1091.255,27.653,442.713,175.263,17.434,152.654
C07957=1091.261,27.903,442.698,175.265,17.435,152.654
C07958=1091.267,28.152,442.684,175.267,17.437,152.654
C07959=1091.273,28.402,442.668,175.269,17.438,152.654
C07960=1091.278,28.651,442.654,175.271,17.440,152.654
C07961=1091.284,28.901,442.638,175.273,17.441,152.654
C07962=1091.290,29.150,442.624,175.274,17.442,152.654
C07963=1091.295,29.399,442.608,175.276,17.445,152.654
C07964=1091.301,29.648,442.593,175.278,17.446,152.654
C07965=1091.306,29.898,442.578,175.279,17.447,152.654
C07966=1091.312,30.148,442.564,175.282,17.449,152.654
C07967=1091.317,30.397,442.549,175.284,17.450,152.654
C07968=1091.324,30.647,442.534,175.285,17.452,152.654
C07969=1091.329,30.896,442.519,175.287,17.453,152.654
C07970=1091.336,31.172,442.502,175.289,17.455,152.654
C07971=1091.342,31.449,442.485,175.291,17.456,152.654
C07972=1091.348,31.725,442.469,175.294,17.458,152.653
C07973=1091.354,32.002,442.452,175.295,17.460,152.654
C07974=1091.361,32.250,442.436,175.297,17.461,152.653
C07975=1091.366,32.500,442.421,175.299,17.462,152.653
C07976=1091.372,32.749,442.406,175.300,17.464,152.653
C07977=1091.378,32.999,442.391,175.303,17.466,152.653
C07978=1091.384,33.249,442.376,175.305,17.467,152.653
C07979=1091.389,33.498,442.361,175.307,17.469,152.653
C07980=1091.395,33.748,442.346,175.308,17.470,152.653
C07981=1091.401,33.997,442.331,175.310,17.471,152.653
C07982=1091.407,34.247,442.316,175.312,17.473,152.653
C07983=1091.412,34.496,442.300,175.314,17.474,152.653
C07984=1091.418,34.746,442.285,175.315,17.476,152.653
C07985=1091.424,34.996,442.270,175.318,17.478,152.653
C07986=1091.429,35.245,442.255,175.319,17.479,152.653
C07987=1091.436,35.494,442.239,175.322,17.480,152.653
C07988=1091.441,35.743,442.224,175.323,17.482,152.653
C07989=1091.447,35.993,442.209,175.325,17.483,152.652
C07990=1091.453,36.243,442.193,175.327,17.485,152.652
C07991=1091.458,36.492,442.178,175.329,17.486,152.652
C07992=1091.464,36.742,442.163,175.331,17.488,152.652
C07993=1091.470,36.990,442.147,175.333,17.489,152.652
C07994=1091.476,37.240,442.132,175.334,17.490,152.652
C07995=1091.482,37.490,442.117,175.337,17.492,152.652
C07996=1091.487,37.739,442.102,175.338,17.494,152.652
C07997=1091.493,37.989,442.087,175.340,17.495,152.652
C07998=1091.499,38.238,442.071,175.342,17.496,152.652
C07999=1091.504,38.487,442.055,175.344,17.498,152.652
C08000=1091.510,38.737,442.040,175.346,17.500,152.652
C08001=1091.515,38.986,442.025,175.348,17.501,152.652
C08002=1091.521,39.236,442.009,175.349,17.502,152.652
C08003=1091.527,39.486,441.993,175.351,17.504,152.652
C08004=1091.533,39.735,441.979,175.353,17.505,152.651
C08005=1091.538,39.985,441.963,175.356,17.507,152.651
C08006=1091.544,40.233,441.947,175.357,17.508,152.651
C08007=1091.549,40.483,441.932,175.359,17.509,152.651
C08008=1091.556,40.733,441.917,175.361,17.511,152.651
C08009=1091.561,40.982,441.901,175.363,17.512,152.651
C08010=1091.567,41.232,441.886,175.365,17.514,152.651
C08011=1091.572,41.482,441.870,175.367,17.515,152.651
C08012=1091.579,41.730,441.855,175.369,17.517,152.651
C08013=1091.584,41.980,441.839,175.371,17.518,152.651
C08014=1091.590,42.230,441.824,175.372,17.520,152.651
C08015=1091.595,42.478,441.808,175.374,17.521,152.651
C08016=1091.601,42.728,441.792,175.376,17.522,152.651
C08017=1091.607,42.978,441.777,175.379,17.524,152.650
C08018=1091.613,43.227,441.761,175.380,17.526,152.650
C08019=1091.618,43.477,441.746,175.382,17.527,152.650
C08020=1091.624,43.727,441.730,175.384,17.528,152.650
C08021=1091.629,43.975,441.714,175.386,17.530,152.650
C08022=1091.635,44.225,441.699,175.388,17.532,152.650
C08023=1091.641,44.475,441.683,175.389,17.533,152.650
C08024=1091.646,44.724,441.667,175.391,17.534,152.650
C08025=1091.653,44.973,441.652,175.394,17.536,152.650
C08026=1091.658,45.223,441.636,175.395,17.537,152.650
C08027=1091.663,45.472,441.621,175.397,17.539,152.650
C08028=1091.669,45.721,441.605,175.399,17.540,152.650
C08029=1091.675,45.971,441.589,175.401,17.542,152.649
C08030=1091.680,46.220,441.573,175.403,17.543,152.650
C08031=1091.686,46.470,441.558,175.404,17.544,152.649
C08032=1091.692,46.719,441.542,175.407,17.546,152.649
C08033=1091.697,46.969,441.526,175.409,17.547,152.649
C08034=1091.703,47.245,441.509,175.411,17.549,152.649
C08035=1091.710,47.522,441.491,175.413,17.551,152.649
C08036=1091.716,47.798,441.474,175.415,17.552,152.649
C08037=1091.722,48.075,441.456,175.417,17.554,152.649
C08038=1091.727,48.323,441.440,175.420,17.556,152.649
C08039=1091.733,48.573,441.424,175.421,17.557,152.649
C08040=1091.738,48.823,441.408,175.423,17.558,152.649
C08041=1091.744,49.072,441.392,175.425,17.560,152.649
C08042=1091.749,49.321,441.377,175.427,17.561,152.648
C08043=1091.755,49.571,441.360,175.429,17.563,152.648
C08044=1091.761,49.821,441.345,175.431,17.564,152.648
C08045=1091.767,50.070,441.329,175.433,17.566,152.648
C08046=1091.772,50.319,441.313,175.435,17.567,152.648
C08047=1091.778,50.569,441.297,175.436,17.568,152.648
C08048=1091.784,50.818,441.281,175.439,17.569,152.648
C08049=1091.790,51.067,441.265,175.440,17.571,152.648
C08050=1091.795,51.317,441.249,175.443,17.573,152.648
C08051=1091.801,51.566,441.233,175.444,17.574,152.648
C08052=1091.807,51.815,441.217,175.447,17.575,152.648
C08053=1091.812,52.065,441.201,175.448,17.576,152.648
C08054=1091.818,52.314,441.186,175.451,17.578,152.647
C08055=1091.824,52.563,441.169,175.453,17.579,152.647
C08056=1091.829,52.813,441.154,175.454,17.580,152.647
C08057=1091.835,53.063,441.137,175.457,17.582,152.647
C08058=1091.841,53.312,441.121,175.458,17.584,152.647
C08059=1091.846,53.562,441.105,175.461,17.585,152.647
C08060=1091.852,53.811,441.089,175.462,17.586,152.647
C08061=1091.858,54.060,441.073,175.465,17.588,152.647
C08062=1091.863,54.310,441.057,175.466,17.589,152.647
C08063=1091.869,54.560,441.041,175.469,17.591,152.647
C08064=1091.875,54.809,441.025,175.470,17.592,152.646
C08065=1091.881,55.058,441.009,175.472,17.593,152.646
C08066=1091.886,55.307,440.993,175.474,17.595,152.646
C08067=1091.892,55.556,440.977,175.476,17.596,152.646
C08068=1091.897,55.807,440.960,175.479,17.597,152.646
C08069=1091.903,56.056,440.944,175.480,17.598,152.646
C08070=1091.909,56.305,440.928,175.483,17.600,152.646
C08071=1091.915,56.555,440.912,175.484,17.601,152.646
C08072=1091.921,56.804,440.895,175.487,17.603,152.646
C08073=1091.927,57.054,440.880,175.488,17.604,152.645
C08074=1091.932,57.303,440.864,175.491,17.606,152.645
C08075=1091.938,57.552,440.848,175.492,17.607,152.645
C08076=1091.943,57.802,440.831,175.494,17.608,152.645
C08077=1091.949,58.051,440.815,175.497,17.609,152.645
C08078=1091.955,58.300,440.798,175.498,17.611,152.645
C08079=1091.961,58.550,440.782,175.501,17.612,152.645
C08080=1091.967,58.799,440.766,175.502,17.613,152.645
C08081=1091.973,59.048,440.750,175.505,17.615,152.645
C08082=1091.978,59.299,440.733,175.506,17.616,152.644
C08083=1091.984,59.548,440.717,175.509,17.618,152.644
C08084=1091.990,59.797,440.701,175.511,17.619,152.644
C08085=1091.996,60.047,440.685,175.513,17.620,152.644
C08086=1092.002,60.296,440.668,175.515,17.622,152.644
C08087=1092.007,60.545,440.652,175.517,17.623,152.644
C08088=1092.012,60.794,440.636,175.519,17.624,152.644
C08089=1092.018,61.044,440.619,175.521,17.626,152.644
C08090=1092.024,61.293,440.603,175.523,17.627,152.644
C08091=1092.030,61.542,440.587,175.524,17.628,152.643
C08092=1092.036,61.792,440.571,175.527,17.630,152.643
C08093=1092.041,62.041,440.554,175.529,17.630,152.643
C08094=1092.047,62.291,440.537,175.531,17.632,152.643
C08095=1092.053,62.540,440.521,175.533,17.633,152.643
C08096=1092.059,62.789,440.505,175.535,17.635,152.643
C08097=1092.064,63.039,440.488,175.537,17.636,152.643
C08098=1092.071,63.315,440.470,175.540,17.638,152.642
C08099=1092.078,63.591,440.452,175.542,17.639,152.642
C08100=1092.084,63.867,440.433,175.544,17.641,152.642
C08101=1092.091,64.144,440.415,175.546,17.641,152.642
C08102=1092.096,64.393,440.399,175.549,17.643,152.642
C08103=1092.103,64.642,440.382,175.550,17.644,152.642
C08104=1092.108,64.892,440.365,175.553,17.646,152.642
C08105=1092.114,65.141,440.349,175.555,17.647,152.642
C08106=1092.120,65.390,440.332,175.557,17.649,152.641
C08107=1092.125,65.640,440.316,175.559,17.650,152.641
C08108=1092.130,65.889,440.300,175.561,17.651,152.641
C08109=1092.136,66.138,440.283,175.563,17.652,152.641
C08110=1092.142,66.388,440.267,175.565,17.654,152.641
C08111=1092.148,66.637,440.250,175.567,17.655,152.641
C08112=1092.154,66.887,440.232,175.570,17.656,152.641
C08113=1092.160,67.136,440.216,175.571,17.657,152.640
C08114=1092.165,67.386,440.199,175.574,17.659,152.640
C08115=1092.171,67.635,440.183,175.575,17.660,152.640
C08116=1092.176,67.884,440.165,175.578,17.662,152.640
C08117=1092.182,68.134,440.149,175.579,17.663,152.640
C08118=1092.187,68.383,440.132,175.582,17.664,152.640
C08119=1092.193,68.633,440.116,175.584,17.665,152.640
C08120=1092.199,68.882,440.099,175.586,17.667,152.639
C08121=1092.205,69.131,440.082,175.588,17.668,152.639
C08122=1092.210,69.381,440.065,175.590,17.670,152.639
C08123=1092.216,69.630,440.049,175.592,17.671,152.639
C08124=1092.222,69.879,440.032,175.595,17.672,152.639
C08125=1092.228,70.128,440.015,175.596,17.673,152.639
C08126=1092.233,70.378,439.998,175.599,17.675,152.639
C08127=1092.239,70.627,439.982,175.600,17.676,152.639
C08128=1092.244,70.876,439.965,175.603,17.677,152.638
C08129=1092.250,71.126,439.948,175.605,17.679,152.638
C08130=1092.255,71.375,439.932,175.607,17.680,152.638
C08131=1092.261,71.625,439.914,175.609,17.681,152.638
C08132=1092.267,71.874,439.898,175.611,17.682,152.638
C08133=1092.272,72.124,439.881,175.613,17.684,152.638
C08134=1092.278,72.372,439.864,175.616,17.685,152.638
C08135=1092.284,72.623,439.847,175.617,17.686,152.637
C08136=1092.290,72.872,439.829,175.620,17.687,152.637
C08137=1092.296,73.121,439.813,175.622,17.689,152.637
C08138=1092.301,73.371,439.796,175.624,17.690,152.637
C08139=1092.306,73.620,439.778,175.626,17.691,152.637
C08140=1092.312,73.869,439.762,175.628,17.692,152.637
C08141=1092.318,74.118,439.745,175.630,17.694,152.637
C08142=1092.324,74.367,439.728,175.632,17.695,152.636
C08143=1092.329,74.617,439.712,175.634,17.696,152.636
C08144=1092.334,74.866,439.694,175.637,17.697,152.636
C08145=1092.341,75.116,439.677,175.638,17.699,152.636
C08146=1092.347,75.365,439.660,175.641,17.700,152.636
C08147=1092.352,75.615,439.643,175.643,17.701,152.636
C08148=1092.358,75.864,439.626,175.645,17.702,152.635
C08149=1092.363,76.113,439.609,175.647,17.704,152.635
C08150=1092.369,76.362,439.592,175.649,17.705,152.635
C08151=1092.375,76.612,439.575,175.651,17.706,152.635
C08152=1092.381,76.861,439.557,175.654,17.708,152.635
C08153=1092.386,77.111,439.540,175.655,17.709,152.635
C08154=1092.392,77.360,439.523,175.658,17.710,152.635
C08155=1092.397,77.609,439.507,175.661,17.711,152.634
C08156=1092.403,77.858,439.489,175.662,17.713,152.634
C08157=1092.409,78.108,439.472,175.665,17.714,152.634
C08158=1092.415,78.358,439.455,175.667,17.715,152.634
C08159=1092.421,78.607,439.437,175.669,17.716,152.634
C08160=1092.426,78.856,439.420,175.671,17.718,152.634
C08161=1092.431,79.105,439.403,175.673,17.719,152.633
C08162=1092.437,79.381,439.384,175.676,17.720,152.633
C08163=1092.443,79.657,439.365,175.678,17.721,152.633
C08164=1092.450,79.934,439.345,175.680,17.723,152.633
C08165=1092.456,80.210,439.327,175.683,17.724,152.633
C08166=1092.462,80.459,439.310,175.684,17.725,152.633
C08167=1092.468,80.708,439.292,175.687,17.727,152.632
C08168=1092.473,80.957,439.275,175.690,17.728,152.632
C08169=1092.478,81.206,439.258,175.691,17.729,152.632
C08170=1092.485,81.456,439.240,175.694,17.730,152.632
C08171=1092.490,81.706,439.223,175.696,17.732,152.632
C08172=1092.495,81.955,439.205,175.698,17.733,152.632
C08173=1092.501,82.204,439.188,175.700,17.734,152.631
C08174=1092.506,82.453,439.170,175.702,17.735,152.631
C08175=1092.513,82.703,439.154,175.704,17.736,152.631
C08176=1092.518,82.952,439.136,175.707,17.738,152.631
C08177=1092.524,83.201,439.118,175.708,17.739,152.631
C08178=1092.529,83.451,439.102,175.711,17.740,152.631
C08179=1092.535,83.701,439.084,175.714,17.742,152.630
C08180=1092.541,83.950,439.066,175.716,17.742,152.630
C08181=1092.546,84.199,439.048,175.718,17.744,152.630
C08182=1092.552,84.448,439.031,175.720,17.745,152.630
C08183=1092.558,84.698,439.014,175.722,17.746,152.630
C08184=1092.563,84.947,438.996,175.724,17.747,152.630
C08185=1092.569,85.196,438.979,175.727,17.748,152.629
C08186=1092.574,85.445,438.961,175.728,17.750,152.629
C08187=1092.580,85.695,438.943,175.731,17.751,152.629
C08188=1092.586,85.945,438.926,175.734,17.752,152.629
C08189=1092.591,86.194,438.909,175.735,17.753,152.629
C08190=1092.597,86.443,438.891,175.738,17.755,152.628
C08191=1092.603,86.692,438.873,175.740,17.755,152.628
C08192=1092.609,86.941,438.856,175.742,17.757,152.628
C08193=1092.614,87.190,438.839,175.744,17.757,152.628
C08194=1092.621,87.440,438.821,175.747,17.759,152.628
C08195=1092.626,87.689,438.803,175.749,17.760,152.628
C08196=1092.632,87.938,438.786,175.751,17.761,152.627
C08197=1092.637,88.188,438.768,175.754,17.763,152.627
C08198=1092.643,88.437,438.751,175.755,17.764,152.627
C08199=1092.648,88.686,438.733,175.758,17.765,152.627
C08200=1092.655,88.936,438.715,175.760,17.766,152.627
C08201=1092.660,89.185,438.698,175.763,17.767,152.626
C08202=1092.666,89.434,438.680,175.764,17.768,152.626
C08203=1092.672,89.684,438.662,175.767,17.769,152.626
C08204=1092.677,89.933,438.645,175.770,17.771,152.626
C08205=1092.682,90.182,438.626,175.771,17.772,152.626
C08206=1092.688,90.432,438.609,175.774,17.773,152.625
C08207=1092.694,90.681,438.591,175.776,17.774,152.625
C08208=1092.700,90.931,438.573,175.778,17.775,152.625
C08209=1092.705,91.180,438.555,175.780,17.776,152.625
C08210=1092.711,91.429,438.538,175.783,17.777,152.625
C08211=1092.717,91.679,438.520,175.785,17.779,152.625
C08212=1092.722,91.928,438.502,175.787,17.780,152.624
C08213=1092.727,92.177,438.484,175.790,17.781,152.624
C08214=1092.734,92.426,438.466,175.792,17.782,152.624
C08215=1092.739,92.675,438.448,175.794,17.783,152.624
C08216=1092.745,92.924,438.430,175.796,17.784,152.624
C08217=1092.751,93.174,438.413,175.799,17.785,152.623
C08218=1092.756,93.423,438.394,175.801,17.787,152.623
C08219=1092.761,93.672,438.377,175.803,17.788,152.623
C08220=1092.767,93.922,438.359,175.806,17.789,152.623
C08221=1092.773,94.171,438.341,175.807,17.790,152.623
C08222=1092.778,94.420,438.324,175.810,17.791,152.622
C08223=1092.784,94.670,438.304,175.813,17.793,152.622
C08224=1092.790,94.919,438.287,175.814,17.793,152.622
C08225=1092.796,95.168,438.269,175.817,17.794,152.622
C08226=1092.801,95.444,438.249,175.820,17.796,152.621
C08227=1092.808,95.721,438.229,175.822,17.797,152.621
C08228=1092.814,95.996,438.209,175.824,17.798,152.621
C08229=1092.820,96.273,438.189,175.827,17.799,152.621
C08230=1092.826,96.522,438.171,175.829,17.801,152.621
C08231=1092.832,96.771,438.153,175.831,17.801,152.620
C08232=1092.837,97.021,438.135,175.834,17.802,152.620
C08233=1092.843,97.270,438.117,175.837,17.804,152.620
C08234=1092.849,97.519,438.099,175.839,17.805,152.620
C08235=1092.854,97.769,438.081,175.841,17.806,152.619
C08236=1092.860,98.018,438.063,175.843,17.807,152.619
C08237=1092.865,98.266,438.045,175.846,17.808,152.619
C08238=1092.871,98.516,438.027,175.848,17.809,152.619
C08239=1092.876,98.765,438.009,175.850,17.810,152.619
C08240=1092.883,99.015,437.990,175.853,17.812,152.618
C08241=1092.888,99.264,437.972,175.855,17.812,152.618
C08242=1092.894,99.514,437.954,175.857,17.813,152.618
C08243=1092.899,99.762,437.936,175.860,17.815,152.618
C08244=1092.906,100.012,437.918,175.862,17.816,152.618
C08245=1092.910,100.261,437.899,175.864,17.817,152.617
C08246=1092.917,100.510,437.881,175.866,17.817,152.617
C08247=1092.922,100.759,437.863,175.869,17.819,152.617
C08248=1092.928,101.009,437.844,175.872,17.820,152.616
C08249=1092.933,101.258,437.826,175.873,17.821,152.616
C08250=1092.940,101.508,437.809,175.876,17.822,152.616
C08251=1092.945,101.756,437.790,175.878,17.823,152.616
C08252=1092.951,102.006,437.772,175.881,17.824,152.616
C08253=1092.956,102.255,437.753,175.883,17.825,152.615
C08254=1092.962,102.505,437.735,175.885,17.826,152.615
C08255=1092.967,102.754,437.717,175.888,17.827,152.615
C08256=1092.973,103.003,437.698,175.890,17.828,152.615
C08257=1092.978,103.252,437.680,175.892,17.830,152.615
C08258=1092.984,103.501,437.661,175.895,17.831,152.614
C08259=1092.989,103.751,437.643,175.897,17.831,152.614
C08260=1092.996,104.000,437.624,175.900,17.832,152.614
C08261=1093.000,104.249,437.606,175.902,17.834,152.614
C08262=1093.007,104.498,437.588,175.904,17.835,152.613
C08263=1093.012,104.748,437.570,175.907,17.836,152.613
C08264=1093.017,104.997,437.550,175.909,17.837,152.613
C08265=1093.023,105.246,437.533,175.911,17.838,152.613
C08266=1093.029,105.496,437.513,175.914,17.839,152.612
C08267=1093.035,105.745,437.495,175.916,17.839,152.612
C08268=1093.040,105.994,437.477,175.919,17.841,152.612
C08269=1093.046,106.243,437.458,175.921,17.842,152.612
C08270=1093.051,106.493,437.440,175.923,17.843,152.612
C08271=1093.057,106.742,437.421,175.926,17.844,152.611
C08272=1093.062,106.991,437.403,175.928,17.845,152.611
C08273=1093.068,107.241,437.384,175.931,17.846,152.611
C08274=1093.074,107.490,437.365,175.933,17.847,152.610
C08275=1093.079,107.739,437.347,175.935,17.848,152.610
C08276=1093.085,107.988,437.328,175.938,17.849,152.610
C08277=1093.091,108.237,437.309,175.941,17.850,152.610
C08278=1093.097,108.487,437.292,175.943,17.851,152.609
C08279=1093.102,108.736,437.272,175.945,17.852,152.609
C08280=1093.107,108.985,437.253,175.948,17.853,152.609
C08281=1093.114,109.235,437.235,175.950,17.854,152.609
C08282=1093.119,109.484,437.216,175.952,17.855,152.609
C08283=1093.125,109.732,437.198,175.954,17.856,152.608
C08284=1093.131,109.982,437.179,175.957,17.857,152.608
C08285=1093.136,110.231,437.161,175.960,17.858,152.608
C08286=1093.142,110.480,437.142,175.962,17.859,152.608
C08287=1093.148,110.730,437.123,175.964,17.860,152.607
C08288=1093.153,110.978,437.104,175.967,17.861,152.607
C08289=1093.159,111.228,437.086,175.969,17.862,152.607
C08290=1093.165,111.504,437.065,175.972,17.862,152.606
C08291=1093.171,111.781,437.044,175.975,17.864,152.606
C08292=1093.178,112.057,437.023,175.977,17.865,152.606
C08293=1093.184,112.333,437.002,175.980,17.866,152.605
C08294=1093.189,112.582,436.984,175.983,17.867,152.605
C08295=1093.195,112.831,436.964,175.985,17.868,152.605
C08296=1093.201,113.080,436.946,175.988,17.869,152.605
C08297=1093.207,113.330,436.926,175.990,17.870,152.604
C08298=1093.212,113.579,436.908,175.992,17.871,152.604
C08299=1093.218,113.828,436.888,175.995,17.872,152.604
C08300=1093.224,114.078,436.870,175.998,17.873,152.604
C08301=1093.229,114.326,436.852,176.000,17.874,152.603
C08302=1093.234,114.576,436.832,176.002,17.875,152.603
C08303=1093.240,114.825,436.813,176.005,17.876,152.603
C08304=1093.245,115.074,436.794,176.007,17.877,152.603
C08305=1093.251,115.324,436.775,176.010,17.878,152.602
C08306=1093.257,115.573,436.756,176.012,17.879,152.602
C08307=1093.262,115.821,436.737,176.014,17.880,152.602
C08308=1093.268,116.071,436.718,176.017,17.881,152.602
C08309=1093.274,116.320,436.699,176.020,17.882,152.601
C08310=1093.279,116.569,436.680,176.022,17.883,152.601
C08311=1093.285,116.818,436.661,176.024,17.884,152.601
C08312=1093.290,117.068,436.642,176.027,17.885,152.601
C08313=1093.295,117.317,436.623,176.029,17.886,152.600
C08314=1093.301,117.566,436.603,176.032,17.887,152.600
C08315=1093.307,117.815,436.584,176.035,17.887,152.600
C08316=1093.312,118.064,436.565,176.037,17.888,152.599
C08317=1093.317,118.314,436.546,176.039,17.889,152.599
C08318=1093.323,118.563,436.527,176.042,17.890,152.599
C08319=1093.329,118.812,436.508,176.044,17.891,152.599
C08320=1093.334,119.061,436.489,176.047,17.892,152.598
C08321=1093.340,119.311,436.469,176.050,17.893,152.598
C08322=1093.345,119.560,436.450,176.051,17.894,152.598
C08323=1093.351,119.809,436.431,176.054,17.895,152.598
C08324=1093.356,120.058,436.412,176.057,17.896,152.597
C08325=1093.362,120.308,436.393,176.059,17.896,152.597
C08326=1093.367,120.557,436.374,176.062,17.898,152.597
C08327=1093.373,120.807,436.354,176.065,17.899,152.596
C08328=1093.379,121.055,436.335,176.066,17.899,152.596
C08329=1093.384,121.304,436.315,176.069,17.901,152.596
C08330=1093.390,121.553,436.296,176.072,17.901,152.595
C08331=1093.396,121.803,436.277,176.074,17.902,152.595
C08332=1093.401,122.052,436.258,176.077,17.903,152.595
C08333=1093.406,122.301,436.239,176.080,17.904,152.595
C08334=1093.412,122.550,436.219,176.081,17.905,152.594
C08335=1093.418,122.799,436.200,176.084,17.906,152.594
C08336=1093.424,123.049,436.180,176.087,17.907,152.594
C08337=1093.429,123.298,436.161,176.090,17.908,152.593
C08338=1093.435,123.547,436.142,176.092,17.909,152.593
C08339=1093.441,123.796,436.122,176.095,17.909,152.593
C08340=1093.446,124.045,436.103,176.098,17.910,152.593
C08341=1093.452,124.295,436.084,176.099,17.911,152.592
C08342=1093.458,124.544,436.065,176.102,17.912,152.592
C08343=1093.464,124.793,436.045,176.105,17.913,152.592
C08344=1093.469,125.043,436.025,176.107,17.914,152.591
C08345=1093.474,125.291,436.006,176.110,17.915,152.591
C08346=1093.480,125.540,435.986,176.113,17.915,152.591
C08347=1093.485,125.790,435.967,176.115,17.916,152.590
C08348=1093.491,126.039,435.948,176.117,17.917,152.590
C08349=1093.497,126.288,435.928,176.120,17.918,152.590
C08350=1093.503,126.537,435.908,176.123,17.919,152.589
C08351=1093.508,126.787,435.889,176.125,17.920,152.589
C08352=1093.514,127.035,435.869,176.128,17.920,152.589
C08353=1093.520,127.285,435.850,176.131,17.922,152.589
C08354=1093.526,127.561,435.828,176.134,17.922,152.588
C08355=1093.532,127.836,435.806,176.136,17.923,152.588
C08356=1093.538,128.113,435.784,176.139,17.924,152.587
C08357=1093.545,128.389,435.763,176.142,17.925,152.587
C08358=1093.550,128.638,435.744,176.144,17.925,152.587
C08359=1093.556,128.887,435.724,176.147,17.927,152.587
C08360=1093.561,129.137,435.704,176.150,17.927,152.586
C08361=1093.567,129.385,435.684,176.152,17.928,152.586
C08362=1093.573,129.635,435.665,176.155,17.929,152.585
C08363=1093.579,129.884,435.645,176.158,17.930,152.585
C08364=1093.584,130.133,435.626,176.161,17.931,152.585
C08365=1093.590,130.382,435.606,176.163,17.931,152.585
C08366=1093.595,130.632,435.586,176.165,17.932,152.584
C08367=1093.601,130.880,435.566,176.168,17.933,152.584
C08368=1093.607,131.130,435.547,176.170,17.934,152.584
C08369=1093.613,131.379,435.527,176.173,17.934,152.583
C08370=1093.619,131.628,435.508,176.176,17.936,152.583
C08371=1093.625,131.877,435.488,176.179,17.936,152.583
C08372=1093.630,132.126,435.467,176.181,17.936,152.582
C08373=1093.636,132.376,435.448,176.184,17.938,152.582
C08374=1093.642,132.624,435.428,176.187,17.939,152.582
C08375=1093.647,132.874,435.408,176.189,17.939,152.581
C08376=1093.653,133.123,435.388,176.192,17.940,152.581
C08377=1093.659,133.372,435.368,176.195,17.941,152.581
C08378=1093.664,133.621,435.348,176.197,17.942,152.580
C08379=1093.670,133.870,435.328,176.199,17.942,152.580
C08380=1093.675,134.119,435.308,176.202,17.943,152.580
C08381=1093.681,134.369,435.288,176.205,17.944,152.579
C08382=1093.687,134.618,435.268,176.208,17.945,152.579
C08383=1093.692,134.867,435.248,176.210,17.945,152.579
C08384=1093.697,135.116,435.229,176.213,17.946,152.578
C08385=1093.703,135.365,435.208,176.216,17.947,152.578
C08386=1093.709,135.614,435.188,176.219,17.948,152.578
C08387=1093.714,135.864,435.169,176.221,17.948,152.577
C08388=1093.720,136.113,435.148,176.223,17.950,152.577
C08389=1093.726,136.362,435.128,176.226,17.950,152.577
C08390=1093.733,136.697,435.102,176.229,17.951,152.576
C08391=1093.741,137.031,435.075,176.233,17.952,152.576
C08392=1093.748,137.366,435.047,176.237,17.954,152.575
C08393=1093.756,137.701,435.020,176.240,17.954,152.575
C08394=1093.762,137.950,435.000,176.243,17.955,152.574
C08395=1093.767,138.199,434.980,176.246,17.956,152.574
C08396=1093.773,138.448,434.960,176.249,17.957,152.574
C08397=1093.778,138.697,434.939,176.251,17.957,152.573
C08398=1093.784,138.946,434.920,176.254,17.958,152.573
C08399=1093.789,139.195,434.900,176.257,17.959,152.573
C08400=1093.795,139.444,434.880,176.260,17.960,152.572
C08401=1093.800,139.693,434.859,176.262,17.960,152.572
C08402=1093.806,139.942,434.839,176.265,17.961,152.572
C08403=1093.812,140.191,434.819,176.268,17.962,152.571
C08404=1093.818,140.440,434.799,176.270,17.963,152.571
C08405=1093.823,140.690,434.778,176.272,17.963,152.571
C08406=1093.829,140.939,434.758,176.275,17.964,152.570
C08407=1093.834,141.189,434.738,176.278,17.965,152.570
C08408=1093.840,141.438,434.717,176.281,17.966,152.569
C08409=1093.846,141.686,434.697,176.284,17.967,152.569
C08410=1093.851,141.936,434.677,176.286,17.967,152.569
C08411=1093.856,142.185,434.656,176.289,17.968,152.568
C08412=1093.862,142.434,434.636,176.292,17.969,152.568
C08413=1093.867,142.683,434.616,176.295,17.969,152.568
C08414=1093.873,142.902,434.598,176.297,17.970,152.567
C08415=1093.877,143.122,434.580,176.299,17.970,152.567
C08416=1093.883,143.342,434.562,176.302,17.971,152.567
C08417=1093.887,143.562,434.544,176.304,17.972,152.566
C08418=1093.892,143.781,434.525,176.306,17.973,152.566
C08419=1093.897,144.001,434.507,176.309,17.973,152.566
C08420=1093.902,144.221,434.489,176.311,17.974,152.566
C08421=1093.907,144.441,434.471,176.314,17.974,152.565
C08422=1093.913,144.691,434.451,176.317,17.975,152.565
C08423=1093.919,144.940,434.431,176.319,17.976,152.564
C08424=1093.924,145.189,434.410,176.321,17.976,152.564
C08425=1093.930,145.437,434.389,176.324,17.977,152.564
C08426=1093.935,145.686,434.369,176.327,17.978,152.563
C08427=1093.941,145.935,434.348,176.330,17.978,152.563
C08428=1093.947,146.185,434.328,176.333,17.980,152.563
C08429=1093.952,146.434,434.307,176.335,17.980,152.562
C08430=1093.958,146.683,434.287,176.338,17.980,152.562
C08431=1093.963,146.932,434.266,176.341,17.981,152.561
C08432=1093.970,147.181,434.245,176.344,17.982,152.561
C08433=1093.975,147.430,434.225,176.346,17.983,152.561
C08434=1093.980,147.679,434.204,176.349,17.983,152.560
C08435=1093.986,147.928,434.183,176.352,17.984,152.560
C08436=1093.992,148.177,434.164,176.355,17.985,152.559
C08437=1093.998,148.426,434.142,176.358,17.985,152.559
C08438=1094.003,148.676,434.121,176.360,17.985,152.559
C08439=1094.008,148.925,434.101,176.363,17.987,152.558
C08440=1094.014,149.174,434.080,176.366,17.987,152.558
C08441=1094.020,149.423,434.059,176.369,17.988,152.558
C08442=1094.026,149.672,434.039,176.372,17.989,152.557
C08443=1094.031,149.921,434.018,176.374,17.989,152.557
C08444=1094.036,150.170,433.998,176.377,17.990,152.556
C08445=1094.042,150.419,433.976,176.380,17.991,152.556
C08446=1094.048,150.668,433.955,176.383,17.992,152.556
C08447=1094.053,150.917,433.935,176.386,17.992,152.555
C08448=1094.058,151.166,433.914,176.388,17.992,152.555
C08449=1094.065,151.415,433.893,176.391,17.993,152.555
C08450=1094.070,151.665,433.873,176.394,17.994,152.554
C08451=1094.076,151.913,433.851,176.397,17.995,152.554
C08452=1094.081,152.162,433.831,176.400,17.996,152.553
C08453=1094.087,152.412,433.810,176.402,17.996,152.553
C08454=1094.093,152.661,433.789,176.405,17.997,152.553
C08455=1094.098,152.910,433.768,176.408,17.997,152.552
C08456=1094.104,153.159,433.746,176.411,17.998,152.552
C08457=1094.109,153.408,433.726,176.414,17.999,152.551
C08458=1094.115,153.657,433.705,176.416,17.999,152.551
C08459=1094.120,153.906,433.684,176.419,18.000,152.551
C08460=1094.126,154.155,433.663,176.422,18.000,152.550
C08461=1094.131,154.404,433.642,176.425,18.001,152.550
C08462=1094.137,154.653,433.621,176.428,18.002,152.549
C08463=1094.143,154.902,433.600,176.431,18.003,152.549
C08464=1094.148,155.151,433.579,176.433,18.003,152.549
C08465=1094.154,155.400,433.558,176.436,18.003,152.548
C08466=1094.160,155.650,433.537,176.439,18.004,152.548
C08467=1094.165,155.898,433.516,176.442,18.005,152.547
C08468=1094.170,156.147,433.495,176.445,18.006,152.547
C08469=1094.177,156.397,433.473,176.447,18.006,152.547
C08470=1094.182,156.645,433.452,176.450,18.006,152.546
C08471=1094.188,156.895,433.431,176.453,18.007,152.546
C08472=1094.194,157.143,433.410,176.456,18.008,152.545
C08473=1094.199,157.393,433.389,176.459,18.009,152.545
C08474=1094.205,157.642,433.368,176.462,18.009,152.544
C08475=1094.210,157.891,433.347,176.464,18.009,152.544
C08476=1094.215,158.140,433.325,176.467,18.010,152.544
C08477=1094.221,158.389,433.304,176.470,18.011,152.543
C08478=1094.226,158.638,433.283,176.473,18.012,152.543
C08479=1094.233,158.887,433.262,176.476,18.012,152.542
C08480=1094.238,159.136,433.240,176.479,18.013,152.542
C08481=1094.243,159.385,433.220,176.482,18.013,152.542
C08482=1094.250,159.661,433.196,176.485,18.014,152.541
C08483=1094.256,159.937,433.172,176.489,18.015,152.541
C08484=1094.262,160.212,433.148,176.492,18.015,152.540
C08485=1094.269,160.488,433.125,176.495,18.016,152.540
C08486=1094.274,160.737,433.104,176.498,18.017,152.539
C08487=1094.280,160.986,433.082,176.501,18.018,152.539
C08488=1094.285,161.235,433.061,176.503,18.017,152.539
C08489=1094.291,161.485,433.040,176.506,18.018,152.538
C08490=1094.297,161.733,433.018,176.509,18.019,152.538
C08491=1094.302,161.982,432.997,176.512,18.019,152.537
C08492=1094.308,162.231,432.975,176.515,18.020,152.537
C08493=1094.313,162.480,432.954,176.518,18.021,152.536
C08494=1094.319,162.729,432.933,176.521,18.022,152.536
C08495=1094.324,162.978,432.911,176.523,18.022,152.536
C08496=1094.329,163.227,432.890,176.526,18.022,152.535
C08497=1094.335,163.476,432.867,176.529,18.023,152.535
C08498=1094.340,163.725,432.846,176.532,18.024,152.534
C08499=1094.346,163.975,432.825,176.535,18.025,152.534
C08500=1094.351,164.223,432.803,176.538,18.025,152.534
C08501=1094.357,164.472,432.782,176.541,18.026,152.533
C08502=1094.362,164.721,432.760,176.544,18.027,152.533
C08503=1094.368,164.970,432.738,176.546,18.027,152.532
C08504=1094.373,165.219,432.716,176.549,18.028,152.532
C08505=1094.379,165.468,432.695,176.552,18.028,152.532
C08506=1094.385,165.717,432.673,176.555,18.029,152.531
C08507=1094.390,165.966,432.651,176.558,18.029,152.531
C08508=1094.396,166.215,432.630,176.561,18.030,152.530
C08509=1094.400,166.464,432.608,176.564,18.031,152.530
C08510=1094.406,166.712,432.587,176.567,18.031,152.529
C08511=1094.411,166.962,432.564,176.570,18.032,152.529
C08512=1094.417,167.210,432.543,176.573,18.032,152.529
C08513=1094.422,167.460,432.521,176.576,18.033,152.528
C08514=1094.428,167.709,432.500,176.579,18.033,152.528
C08515=1094.433,167.958,432.477,176.582,18.034,152.527
C08516=1094.439,168.207,432.456,176.585,18.035,152.527
C08517=1094.444,168.456,432.434,176.588,18.036,152.526
C08518=1094.450,168.705,432.413,176.591,18.036,152.526
C08519=1094.455,168.954,432.390,176.593,18.036,152.526
C08520=1094.462,169.203,432.369,176.596,18.037,152.525
C08521=1094.466,169.452,432.347,176.599,18.037,152.525
C08522=1094.473,169.701,432.325,176.602,18.038,152.524
C08523=1094.477,169.950,432.303,176.605,18.038,152.524
C08524=1094.484,170.199,432.282,176.608,18.039,152.523
C08525=1094.488,170.448,432.260,176.611,18.040,152.523
C08526=1094.495,170.697,432.238,176.614,18.041,152.523
C08527=1094.500,170.946,432.216,176.618,18.041,152.522
C08528=1094.506,171.195,432.194,176.620,18.041,152.522
C08529=1094.511,171.444,432.172,176.623,18.042,152.521
C08530=1094.517,171.693,432.151,176.626,18.042,152.521
C08531=1094.523,171.942,432.128,176.629,18.043,152.520
C08532=1094.527,172.190,432.106,176.632,18.043,152.520
C08533=1094.534,172.440,432.084,176.635,18.044,152.519
C08534=1094.539,172.689,432.062,176.638,18.044,152.519
C08535=1094.545,172.938,432.041,176.641,18.045,152.518
C08536=1094.550,173.187,432.018,176.644,18.046,152.518
C08537=1094.556,173.436,431.996,176.647,18.046,152.518
C08538=1094.561,173.685,431.974,176.650,18.046,152.517
C08539=1094.567,173.934,431.951,176.653,18.047,152.517
C08540=1094.573,174.182,431.930,176.656,18.047,152.516
C08541=1094.578,174.432,431.908,176.659,18.048,152.516
C08542=1094.584,174.681,431.886,176.662,18.048,152.515
C08543=1094.589,174.929,431.864,176.665,18.049,152.515
C08544=1094.595,175.178,431.841,176.668,18.050,152.514
C08545=1094.601,175.427,431.819,176.671,18.050,152.514
C08546=1094.607,175.703,431.795,176.674,18.051,152.513
C08547=1094.613,175.978,431.770,176.678,18.051,152.513
C08548=1094.620,176.253,431.745,176.681,18.051,152.512
C08549=1094.626,176.529,431.721,176.685,18.053,152.512
C08550=1094.631,176.777,431.699,176.688,18.053,152.511
C08551=1094.637,177.027,431.677,176.690,18.053,152.511
C08552=1094.642,177.276,431.655,176.693,18.053,152.510
C08553=1094.648,177.525,431.632,176.696,18.054,152.510
C08554=1094.654,177.773,431.611,176.700,18.054,152.509
C08555=1094.659,178.022,431.588,176.703,18.055,152.509
C08556=1094.665,178.272,431.565,176.706,18.055,152.508
C08557=1094.671,178.520,431.543,176.709,18.056,152.508
C08558=1094.676,178.769,431.521,176.712,18.056,152.507
C08559=1094.682,179.018,431.498,176.715,18.057,152.507
C08560=1094.688,179.267,431.477,176.718,18.057,152.507
C08561=1094.694,179.516,431.454,176.721,18.058,152.506
C08562=1094.699,179.765,431.432,176.725,18.058,152.506
C08563=1094.705,180.014,431.409,176.728,18.059,152.505
C08564=1094.711,180.263,431.386,176.730,18.059,152.505
C08565=1094.716,180.512,431.364,176.733,18.059,152.504
C08566=1094.722,180.761,431.341,176.736,18.060,152.504
C08567=1094.728,181.009,431.320,176.739,18.060,152.503
C08568=1094.733,181.258,431.297,176.742,18.061,152.503
C08569=1094.739,181.507,431.274,176.746,18.061,152.502
C08570=1094.745,181.756,431.252,176.749,18.062,152.502
C08571=1094.751,182.005,431.230,176.752,18.062,152.501
C08572=1094.757,182.254,431.207,176.755,18.062,152.501
C08573=1094.762,182.504,431.184,176.758,18.063,152.500
C08574=1094.768,182.752,431.162,176.761,18.063,152.500
C08575=1094.774,183.001,431.139,176.764,18.064,152.499
C08576=1094.779,183.250,431.117,176.768,18.064,152.499
C08577=1094.785,183.499,431.094,176.771,18.064,152.498
C08578=1094.791,183.748,431.071,176.774,18.065,152.498
C08579=1094.797,183.996,431.049,176.777,18.065,152.497
C08580=1094.802,184.246,431.027,176.780,18.065,152.497
C08581=1094.808,184.495,431.004,176.783,18.066,152.496
C08582=1094.813,184.743,430.981,176.786,18.066,152.496
C08583=1094.820,184.992,430.959,176.789,18.066,152.495
C08584=1094.825,185.241,430.937,176.792,18.067,152.495
C08585=1094.831,185.490,430.914,176.795,18.067,152.494
C08586=1094.836,185.739,430.890,176.798,18.068,152.494
C08587=1094.842,185.988,430.867,176.802,18.068,152.493
C08588=1094.847,186.236,430.845,176.805,18.069,152.493
C08589=1094.852,186.486,430.822,176.808,18.070,152.492
C08590=1094.858,186.735,430.799,176.811,18.070,152.492
C08591=1094.864,186.984,430.776,176.814,18.071,152.491
C08592=1094.869,187.233,430.754,176.817,18.071,152.491
C08593=1094.875,187.481,430.731,176.820,18.072,152.490
C08594=1094.880,187.730,430.708,176.823,18.072,152.490
C08595=1094.885,187.979,430.684,176.826,18.073,152.489
C08596=1094.891,188.228,430.662,176.829,18.073,152.489
C08597=1094.896,188.477,430.639,176.833,18.074,152.489
C08598=1094.902,188.726,430.616,176.836,18.074,152.488
C08599=1094.908,188.975,430.593,176.839,18.075,152.488
C08600=1094.913,189.223,430.571,176.842,18.075,152.487
C08601=1094.919,189.472,430.548,176.845,18.076,152.487
C08602=1094.924,189.721,430.524,176.848,18.076,152.486
C08603=1094.929,189.970,430.501,176.852,18.076,152.486
C08604=1094.935,190.219,430.478,176.855,18.077,152.485
C08605=1094.941,190.468,430.455,176.858,18.077,152.485
C08606=1094.947,190.717,430.433,176.861,18.078,152.484
C08607=1094.952,190.966,430.409,176.864,18.078,152.484
C08608=1094.957,191.215,430.386,176.867,18.078,152.483
C08609=1094.962,191.463,430.363,176.870,18.079,152.483
C08610=1094.969,191.738,430.338,176.874,18.079,152.482
C08611=1094.975,192.013,430.312,176.877,18.080,152.482
C08612=1094.982,192.288,430.287,176.881,18.081,152.481
C08613=1094.988,192.564,430.261,176.884,18.081,152.480
C08614=1094.993,192.812,430.238,176.887,18.081,152.480
C08615=1094.999,193.061,430.215,176.890,18.082,152.479
C08616=1095.004,193.311,430.191,176.894,18.082,152.479
C08617=1095.010,193.559,430.168,176.897,18.082,152.478
C08618=1095.016,193.808,430.145,176.900,18.083,152.478
C08619=1095.022,194.057,430.122,176.903,18.083,152.477
C08620=1095.027,194.306,430.098,176.906,18.084,152.477
C08621=1095.032,194.555,430.075,176.910,18.084,152.476
C08622=1095.038,194.804,430.052,176.913,18.085,152.476
C08623=1095.044,195.053,430.029,176.916,18.085,152.475
C08624=1095.049,195.301,430.005,176.919,18.085,152.475
C08625=1095.055,195.550,429.982,176.922,18.086,152.474
C08626=1095.061,195.799,429.959,176.925,18.086,152.474
C08627=1095.066,196.048,429.936,176.929,18.087,152.473
C08628=1095.072,196.296,429.912,176.932,18.087,152.473
C08629=1095.077,196.545,429.889,176.935,18.087,152.472
C08630=1095.083,196.794,429.866,176.938,18.088,152.472
C08631=1095.088,197.043,429.842,176.941,18.088,152.471
C08632=1095.094,197.292,429.819,176.945,18.089,152.471
C08633=1095.100,197.541,429.796,176.948,18.089,152.470
C08634=1095.105,197.789,429.772,176.951,18.089,152.470
C08635=1095.111,198.038,429.749,176.954,18.089,152.469
C08636=1095.117,198.287,429.726,176.957,18.090,152.469
C08637=1095.122,198.536,429.701,176.961,18.090,152.468
C08638=1095.128,198.785,429.678,176.964,18.091,152.468
C08639=1095.134,199.033,429.654,176.967,18.091,152.467
C08640=1095.139,199.283,429.631,176.970,18.091,152.467
C08641=1095.145,199.531,429.608,176.974,18.092,152.466
C08642=1095.151,199.780,429.584,176.977,18.092,152.465
C08643=1095.156,200.029,429.561,176.981,18.093,152.465
C08644=1095.162,200.277,429.537,176.984,18.094,152.464
C08645=1095.168,200.526,429.514,176.987,18.094,152.464
C08646=1095.174,200.775,429.489,176.990,18.094,152.463
C08647=1095.179,201.024,429.467,176.994,18.094,152.463
C08648=1095.185,201.273,429.442,176.997,18.095,152.462
C08649=1095.190,201.522,429.419,177.000,18.095,152.462
C08650=1095.197,201.770,429.396,177.003,18.095,152.461
C08651=1095.202,202.019,429.372,177.007,18.096,152.461
C08652=1095.208,202.268,429.348,177.010,18.096,152.460
C08653=1095.213,202.517,429.325,177.013,18.097,152.460
C08654=1095.219,202.766,429.301,177.016,18.097,152.459
C08655=1095.224,203.014,429.277,177.019,18.097,152.459
C08656=1095.230,203.263,429.254,177.022,18.097,152.458
C08657=1095.236,203.512,429.229,177.026,18.098,152.457
C08658=1095.242,203.761,429.206,177.029,18.098,152.457
C08659=1095.247,204.010,429.182,177.032,18.098,152.456
C08660=1095.252,204.259,429.158,177.035,18.099,152.456
C08661=1095.258,204.508,429.135,177.038,18.099,152.455
C08662=1095.263,204.756,429.110,177.042,18.100,152.455
C08663=1095.269,205.004,429.087,177.046,18.101,152.454
C08664=1095.275,205.254,429.063,177.049,18.101,152.454
C08665=1095.280,205.503,429.039,177.052,18.101,152.453
C08666=1095.286,205.751,429.015,177.055,18.101,152.453
C08667=1095.292,206.000,428.991,177.058,18.102,152.452
C08668=1095.297,206.249,428.967,177.062,18.102,152.452
C08669=1095.303,206.498,428.943,177.065,18.103,152.451
C08670=1095.309,206.747,428.919,177.068,18.103,152.451
C08671=1095.314,206.995,428.895,177.071,18.103,152.450
C08672=1095.320,207.244,428.872,177.075,18.104,152.450
C08673=1095.326,207.493,428.847,177.078,18.104,152.449
C08674=1095.348,208.507,428.749,177.131,18.126,152.444
C08675=1095.357,208.881,428.713,177.136,18.128,152.443
C08676=1095.365,209.255,428.676,177.140,18.130,152.443
C08677=1095.374,209.629,428.640,177.145,18.132,152.443
C08678=1095.382,210.002,428.602,177.150,18.134,152.442
C08679=1095.388,210.251,428.578,177.153,18.135,152.442
C08680=1095.394,210.500,428.554,177.156,18.137,152.441
C08681=1095.399,210.748,428.530,177.159,18.138,152.441
C08682=1095.405,210.998,428.505,177.162,18.139,152.441
C08683=1095.410,211.246,428.481,177.165,18.140,152.441
C08684=1095.416,211.495,428.457,177.168,18.141,152.440
C08685=1095.421,211.744,428.432,177.172,18.143,152.440
C08686=1095.427,211.993,428.408,177.174,18.144,152.440
C08687=1095.433,212.241,428.383,177.177,18.145,152.439
C08688=1095.438,212.490,428.358,177.181,18.147,152.439
C08689=1095.444,212.738,428.334,177.184,18.148,152.439
C08690=1095.449,212.988,428.309,177.187,18.149,152.438
C08691=1095.455,213.236,428.285,177.190,18.151,152.438
C08692=1095.461,213.485,428.260,177.193,18.151,152.438
C08693=1095.466,213.734,428.236,177.197,18.153,152.437
C08694=1095.472,213.982,428.211,177.200,18.154,152.437
C08695=1095.477,214.231,428.187,177.202,18.155,152.437
C08696=1095.483,214.479,428.162,177.206,18.157,152.437
C08697=1095.489,214.729,428.137,177.209,18.158,152.436
C08698=1095.494,214.977,428.113,177.212,18.159,152.436
C08699=1095.500,215.226,428.087,177.215,18.161,152.436
C08700=1095.505,215.475,428.063,177.218,18.161,152.435
C08701=1095.510,215.723,428.038,177.222,18.163,152.435
C08702=1095.517,215.972,428.013,177.224,18.165,152.435
C08703=1095.522,216.221,427.989,177.228,18.166,152.434
C08704=1095.528,216.470,427.964,177.231,18.167,152.434
C08705=1095.533,216.718,427.939,177.235,18.168,152.434
C08706=1095.539,216.967,427.915,177.237,18.170,152.433
C08707=1095.544,217.216,427.889,177.240,18.171,152.433
C08708=1095.550,217.465,427.864,177.244,18.172,152.433
C08709=1095.556,217.713,427.839,177.247,18.173,152.433
C08710=1095.562,217.962,427.815,177.250,18.175,152.432
C08711=1095.567,218.211,427.791,177.253,18.176,152.432
C08712=1095.573,218.459,427.765,177.256,18.177,152.432
C08713=1095.578,218.708,427.740,177.260,18.179,152.431
C08714=1095.584,218.957,427.715,177.262,18.180,152.431
C08715=1095.589,219.205,427.691,177.266,18.182,152.431
C08716=1095.595,219.454,427.665,177.269,18.182,152.430
C08717=1095.601,219.702,427.641,177.272,18.184,152.430
C08718=1095.606,219.952,427.615,177.275,18.185,152.430
C08719=1095.612,220.200,427.590,177.278,18.186,152.429
C08720=1095.618,220.449,427.566,177.282,18.188,152.429
C08721=1095.624,220.698,427.540,177.285,18.189,152.429
C08722=1095.628,220.947,427.516,177.288,18.191,152.429
C08723=1095.635,221.195,427.490,177.291,18.192,152.428
C08724=1095.641,221.444,427.465,177.295,18.193,152.428
C08725=1095.646,221.692,427.441,177.297,18.194,152.428
C08726=1095.652,221.941,427.415,177.301,18.196,152.427
C08727=1095.661,222.319,427.377,177.306,18.198,152.427
C08728=1095.668,222.696,427.339,177.310,18.200,152.426
C08729=1095.677,223.074,427.300,177.315,18.201,152.426
C08730=1095.686,223.451,427.262,177.319,18.203,152.426
C08731=1095.691,223.700,427.236,177.323,18.205,152.425
C08732=1095.697,223.948,427.212,177.326,18.206,152.425
C08733=1095.702,224.198,427.186,177.330,18.208,152.425
C08734=1095.708,224.446,427.161,177.332,18.209,152.424
C08735=1095.713,224.695,427.135,177.336,18.211,152.424
C08736=1095.719,224.944,427.110,177.339,18.212,152.424
C08737=1095.725,225.191,427.085,177.342,18.213,152.423
C08738=1095.730,225.441,427.060,177.345,18.215,152.423
C08739=1095.736,225.690,427.035,177.349,18.216,152.423
C08740=1095.741,225.938,427.009,177.351,18.217,152.423
C08741=1095.747,226.187,426.984,177.355,18.219,152.422
C08742=1095.753,226.436,426.958,177.358,18.220,152.422
C08743=1095.758,226.684,426.933,177.361,18.222,152.422
C08744=1095.764,226.933,426.907,177.364,18.223,152.421
C08745=1095.770,227.181,426.881,177.368,18.224,152.421
C08746=1095.775,227.430,426.857,177.371,18.225,152.421
C08747=1095.781,227.679,426.831,177.373,18.227,152.421
C08748=1095.786,227.928,426.805,177.377,18.228,152.420
C08749=1095.792,228.177,426.780,177.380,18.229,152.420
C08750=1095.797,228.425,426.754,177.383,18.231,152.420
C08751=1095.804,228.673,426.729,177.386,18.232,152.419
C08752=1095.809,228.922,426.703,177.390,18.234,152.419
C08753=1095.815,229.170,426.678,177.393,18.235,152.419
C08754=1095.820,229.419,426.652,177.396,18.236,152.418
C08755=1095.826,229.668,426.626,177.399,18.237,152.418
C08756=1095.832,229.917,426.601,177.403,18.239,152.418
C08757=1095.838,230.165,426.574,177.406,18.240,152.417
C08758=1095.843,230.413,426.549,177.409,18.242,152.417
C08759=1095.849,230.662,426.523,177.412,18.243,152.417
C08760=1095.854,230.911,426.497,177.416,18.244,152.417
C08761=1095.860,231.160,426.472,177.418,18.246,152.416
C08762=1095.865,231.408,426.447,177.422,18.247,152.416
C08763=1095.871,231.657,426.421,177.425,18.249,152.416
C08764=1095.877,231.906,426.395,177.428,18.250,152.415
C08765=1095.882,232.155,426.369,177.431,18.251,152.415
C08766=1095.887,232.403,426.343,177.435,18.253,152.415
C08767=1095.894,232.651,426.318,177.438,18.254,152.415
C08768=1095.899,232.900,426.292,177.441,18.256,152.414
C08769=1095.905,233.149,426.266,177.444,18.257,152.414
C08770=1095.910,233.398,426.240,177.447,18.259,152.414
C08771=1095.916,233.646,426.214,177.450,18.260,152.413
C08772=1095.921,233.895,426.188,177.454,18.261,152.413
C08773=1095.927,234.143,426.162,177.457,18.263,152.413
C08774=1095.933,234.392,426.136,177.460,18.264,152.413
C08775=1095.938,234.641,426.110,177.464,18.266,152.412
C08776=1095.944,234.889,426.085,177.467,18.267,152.412
C08777=1095.949,235.138,426.059,177.470,18.269,152.412
C08778=1095.955,235.386,426.032,177.473,18.270,152.412
C08779=1095.964,235.756,425.994,177.477,18.272,152.411
C08780=1095.972,236.125,425.955,177.483,18.274,152.411
C08781=1095.980,236.493,425.916,177.487,18.276,152.410
C08782=1095.988,236.862,425.877,177.492,18.278,152.410
C08783=1095.994,237.111,425.852,177.496,18.280,152.410
C08784=1096.000,237.360,425.826,177.498,18.281,152.409
C08785=1096.005,237.608,425.799,177.502,18.283,152.409
C08786=1096.011,237.857,425.773,177.505,18.284,152.409
C08787=1096.017,238.105,425.747,177.508,18.286,152.408
C08788=1096.022,238.354,425.721,177.511,18.287,152.408
C08789=1096.027,238.602,425.694,177.515,18.289,152.408
C08790=1096.033,238.851,425.668,177.518,18.290,152.408
C08791=1096.038,239.099,425.642,177.521,18.291,152.407
C08792=1096.044,239.348,425.616,177.525,18.293,152.407
C08793=1096.050,239.597,425.589,177.527,18.294,152.407
C08794=1096.056,239.845,425.564,177.531,18.296,152.406
C08795=1096.062,240.094,425.537,177.534,18.297,152.406
C08796=1096.067,240.342,425.511,177.537,18.299,152.406
C08797=1096.073,240.591,425.485,177.541,18.301,152.406
C08798=1096.079,240.839,425.458,177.544,18.301,152.405
C08799=1096.084,241.088,425.432,177.547,18.303,152.405
C08800=1096.090,241.337,425.405,177.550,18.304,152.405
C08801=1096.096,241.585,425.379,177.554,18.306,152.405
C08802=1096.101,241.834,425.353,177.557,18.307,152.404
C08803=1096.107,242.082,425.326,177.560,18.309,152.404
C08804=1096.113,242.331,425.300,177.563,18.310,152.404
C08805=1096.118,242.580,425.274,177.566,18.312,152.404
C08806=1096.124,242.828,425.247,177.570,18.313,152.403
C08807=1096.129,243.077,425.220,177.573,18.315,152.403
C08808=1096.135,243.325,425.193,177.576,18.316,152.403
C08809=1096.140,243.574,425.167,177.579,18.318,152.402
C08810=1096.146,243.823,425.141,177.583,18.319,152.402
C08811=1096.152,244.071,425.114,177.586,18.321,152.402
C08812=1096.158,244.319,425.087,177.589,18.322,152.402
C08813=1096.163,244.568,425.061,177.593,18.324,152.401
C08814=1096.168,244.817,425.034,177.595,18.325,152.401
C08815=1096.174,245.065,425.007,177.599,18.327,152.401
C08816=1096.180,245.314,424.981,177.602,18.329,152.401
C08817=1096.185,245.562,424.954,177.605,18.330,152.400
C08818=1096.191,245.810,424.927,177.609,18.332,152.400
C08819=1096.196,246.059,424.900,177.611,18.333,152.400
C08820=1096.202,246.307,424.874,177.615,18.334,152.399
C08821=1096.207,246.556,424.848,177.619,18.336,152.399
C08822=1096.213,246.805,424.821,177.621,18.337,152.399
C08823=1096.218,247.053,424.794,177.625,18.339,152.399
C08824=1096.224,247.302,424.767,177.627,18.341,152.398
C08825=1096.230,247.550,424.740,177.631,18.342,152.398
C08826=1096.235,247.799,424.713,177.635,18.344,152.398
C08827=1096.241,248.047,424.687,177.637,18.345,152.398
C08828=1096.246,248.295,424.660,177.641,18.347,152.397
C08829=1096.251,248.544,424.633,177.645,18.349,152.397
C08830=1096.257,248.793,424.606,177.647,18.350,152.397
C08831=1096.266,249.194,424.563,177.652,18.353,152.397
C08832=1096.275,249.595,424.519,177.658,18.355,152.396
C08833=1096.284,249.996,424.475,177.663,18.358,152.396
C08834=1096.293,250.397,424.431,177.668,18.361,152.395
C08835=1096.299,250.646,424.405,177.671,18.362,152.395
C08836=1096.304,250.894,424.377,177.675,18.364,152.395
C08837=1096.310,251.143,424.351,177.677,18.365,152.395
C08838=1096.315,251.391,424.323,177.681,18.367,152.394
C08839=1096.321,251.639,424.296,177.685,18.368,152.394
C08840=1096.326,251.888,424.269,177.687,18.369,152.394
C08841=1096.332,252.137,424.242,177.691,18.371,152.394
C08842=1096.338,252.385,424.215,177.694,18.373,152.393
C08843=1096.343,252.633,424.187,177.697,18.374,152.393
C08844=1096.349,252.882,424.161,177.701,18.376,152.393
C08845=1096.354,253.130,424.133,177.704,18.378,152.393
C08846=1096.360,253.379,424.107,177.707,18.379,152.392
C08847=1096.365,253.608,424.081,177.710,18.381,152.392
C08848=1096.371,253.837,424.056,177.713,18.382,152.392
C08849=1096.375,254.066,424.031,177.716,18.384,152.392
C08850=1096.381,254.294,424.006,177.719,18.385,152.391
C08851=1096.386,254.524,423.981,177.722,18.387,152.391
C08852=1096.391,254.753,423.955,177.726,18.388,152.391
C08853=1096.396,254.981,423.930,177.728,18.390,152.391
C08854=1096.402,255.211,423.904,177.731,18.391,152.391
C08855=1096.407,255.459,423.878,177.734,18.393,152.390
C08856=1096.412,255.708,423.851,177.738,18.395,152.390
C08857=1096.419,255.955,423.823,177.741,18.396,152.390
C08858=1096.424,256.204,423.796,177.744,18.398,152.390
C08859=1096.430,256.453,423.768,177.748,18.399,152.389
C08860=1096.435,256.701,423.741,177.750,18.401,152.389
C08861=1096.441,256.949,423.713,177.754,18.403,152.389
C08862=1096.447,257.198,423.686,177.757,18.404,152.389
C08863=1096.452,257.446,423.658,177.760,18.406,152.388
C08864=1096.458,257.695,423.631,177.764,18.407,152.388
C08865=1096.463,257.943,423.603,177.767,18.409,152.388
C08866=1096.469,258.192,423.576,177.770,18.411,152.388
C08867=1096.475,258.440,423.549,177.773,18.412,152.387
C08868=1096.480,258.689,423.521,177.777,18.414,152.387
C08869=1096.487,258.937,423.494,177.780,18.415,152.387
C08870=1096.492,259.186,423.466,177.783,18.417,152.387
C08871=1096.497,259.434,423.438,177.787,18.419,152.387
C08872=1096.504,259.682,423.411,177.789,18.420,152.386
C08873=1096.509,259.931,423.383,177.793,18.422,152.386
C08874=1096.514,260.179,423.355,177.796,18.424,152.386
C08875=1096.521,260.427,423.328,177.799,18.425,152.385
C08876=1096.526,260.676,423.300,177.803,18.427,152.385
C08877=1096.532,260.925,423.272,177.806,18.428,152.385
C08878=1096.538,261.173,423.245,177.810,18.430,152.385
C08879=1096.543,261.421,423.217,177.813,18.431,152.385
C08880=1096.549,261.670,423.189,177.816,18.433,152.384
C08881=1096.555,261.918,423.162,177.820,18.435,152.384
C08882=1096.561,262.166,423.133,177.822,18.436,152.384
C08883=1096.569,262.526,423.094,177.828,18.439,152.384
C08884=1096.577,262.885,423.054,177.832,18.441,152.383
C08885=1096.585,263.245,423.013,177.837,18.444,152.383
C08886=1096.594,263.603,422.973,177.842,18.446,152.382
C08887=1096.600,263.852,422.945,177.845,18.447,152.382
C08888=1096.606,264.100,422.918,177.848,18.449,152.382
C08889=1096.611,264.348,422.890,177.852,18.451,152.382
C08890=1096.617,264.597,422.861,177.855,18.453,152.381
C08891=1096.622,264.845,422.833,177.858,18.454,152.381
C08892=1096.628,265.094,422.805,177.861,18.456,152.381
C08893=1096.633,265.342,422.778,177.865,18.458,152.381
C08894=1096.639,265.591,422.749,177.868,18.460,152.381
C08895=1096.645,265.839,422.721,177.871,18.461,152.380
C08896=1096.651,266.087,422.694,177.874,18.463,152.380
C08897=1096.657,266.335,422.666,177.878,18.465,152.380
C08898=1096.662,266.584,422.638,177.881,18.466,152.380
C08899=1096.668,266.832,422.609,177.884,18.468,152.380
C08900=1096.673,267.080,422.581,177.887,18.470,152.379
C08901=1096.679,267.329,422.553,177.891,18.472,152.379
C08902=1096.684,267.577,422.525,177.894,18.473,152.379
C08903=1096.690,267.826,422.497,177.897,18.475,152.379
C08904=1096.696,268.074,422.469,177.901,18.477,152.379
C08905=1096.702,268.322,422.440,177.904,18.479,152.378
C08906=1096.707,268.570,422.412,177.907,18.480,152.378
C08907=1096.713,268.818,422.384,177.910,18.482,152.378
C08908=1096.719,269.067,422.356,177.914,18.484,152.378
C08909=1096.725,269.316,422.327,177.917,18.486,152.377
C08910=1096.730,269.564,422.299,177.920,18.487,152.377
C08911=1096.735,269.813,422.270,177.924,18.489,152.377
C08912=1096.741,270.060,422.242,177.927,18.491,152.377
C08913=1096.747,270.309,422.213,177.930,18.493,152.377
C08914=1096.752,270.557,422.185,177.933,18.495,152.377
C08915=1096.758,270.806,422.157,177.937,18.496,152.376
C08916=1096.763,271.054,422.129,177.940,18.498,152.376
C08917=1096.770,271.302,422.100,177.944,18.500,152.376
C08918=1096.775,271.550,422.072,177.947,18.502,152.376
C08919=1096.781,271.799,422.044,177.950,18.504,152.375
C08920=1096.786,272.046,422.015,177.953,18.505,152.375
C08921=1096.792,272.295,421.986,177.957,18.507,152.375
C08922=1096.797,272.543,421.958,177.960,18.509,152.375
C08923=1096.803,272.792,421.930,177.963,18.511,152.375
C08924=1096.809,273.040,421.901,177.966,18.513,152.374
C08925=1096.814,273.289,421.872,177.970,18.514,152.374
C08926=1096.820,273.537,421.843,177.973,18.517,152.374
C08927=1096.825,273.785,421.815,177.976,18.519,152.374
C08928=1096.831,274.033,421.787,177.979,18.520,152.374
C08929=1096.838,274.282,421.758,177.983,18.522,152.373
C08930=1096.842,274.530,421.729,177.986,18.524,152.373
C08931=1096.848,274.778,421.700,177.989,18.526,152.373
C08932=1096.854,275.026,421.672,177.992,18.527,152.373
C08933=1096.859,275.275,421.643,177.995,18.529,152.373
C08934=1096.865,275.523,421.615,177.999,18.531,152.373
C08935=1096.873,275.885,421.573,178.004,18.534,152.372
C08936=1096.881,276.246,421.531,178.008,18.536,152.372
C08937=1096.890,276.609,421.489,178.013,18.539,152.372
C08938=1096.898,276.970,421.447,178.018,18.542,152.372
C08939=1096.904,277.219,421.418,178.021,18.544,152.371
C08940=1096.910,277.467,421.389,178.025,18.546,152.371
C08941=1096.914,277.716,421.361,178.028,18.548,152.371
C08942=1096.921,277.964,421.332,178.032,18.550,152.371
C08943=1096.926,278.211,421.303,178.034,18.551,152.371
C08944=1096.931,278.460,421.274,178.038,18.553,152.371
C08945=1096.938,278.709,421.245,178.041,18.555,152.370
C08946=1096.943,278.957,421.215,178.044,18.557,152.370
C08947=1096.949,279.205,421.187,178.048,18.559,152.370
C08948=1096.955,279.453,421.158,178.050,18.561,152.370
C08949=1096.960,279.702,421.129,178.054,18.563,152.370
C08950=1096.966,279.949,421.100,178.057,18.564,152.369
C08951=1096.971,280.198,421.071,178.061,18.567,152.369
C08952=1096.977,280.446,421.042,178.064,18.569,152.369
C08953=1096.983,280.695,421.012,178.067,18.571,152.369
C08954=1096.989,280.942,420.984,178.070,18.572,152.369
C08955=1096.994,281.191,420.955,178.074,18.574,152.369
C08956=1097.000,281.439,420.926,178.077,18.576,152.369
C08957=1097.005,281.687,420.897,178.080,18.578,152.368
C08958=1097.011,281.935,420.867,178.084,18.580,152.368
C08959=1097.017,282.184,420.838,178.087,18.582,152.368
C08960=1097.022,282.432,420.808,178.090,18.584,152.368
C08961=1097.028,282.680,420.780,178.093,18.586,152.368
C08962=1097.033,282.929,420.751,178.096,18.588,152.368
C08963=1097.039,283.177,420.722,178.100,18.590,152.367
C08964=1097.045,283.425,420.692,178.103,18.592,152.367
C08965=1097.050,283.673,420.663,178.106,18.594,152.367
C08966=1097.056,283.921,420.634,178.110,18.596,152.367
C08967=1097.062,284.169,420.604,178.112,18.598,152.367
C08968=1097.067,284.418,420.574,178.116,18.600,152.367
C08969=1097.073,284.665,420.546,178.119,18.602,152.367
C08970=1097.078,284.914,420.516,178.123,18.604,152.366
C08971=1097.084,285.162,420.486,178.126,18.606,152.366
C08972=1097.090,285.410,420.457,178.130,18.608,152.366
C08973=1097.095,285.659,420.428,178.133,18.610,152.366
C08974=1097.100,285.907,420.398,178.136,18.612,152.366
C08975=1097.107,286.155,420.369,178.139,18.614,152.366
C08976=1097.112,286.403,420.340,178.142,18.616,152.365
C08977=1097.118,286.652,420.310,178.146,18.618,152.365
C08978=1097.124,286.899,420.280,178.149,18.620,152.365
C08979=1097.130,287.147,420.251,178.152,18.622,152.365
C08980=1097.135,287.395,420.222,178.156,18.624,152.365
C08981=1097.140,287.644,420.192,178.159,18.626,152.365
C08982=1097.146,287.892,420.163,178.162,18.628,152.365
C08983=1097.152,288.140,420.133,178.165,18.630,152.365
C08984=1097.158,288.388,420.103,178.168,18.632,152.364
C08985=1097.164,288.636,420.074,178.172,18.634,152.364
C08986=1097.169,288.885,420.044,178.175,18.636,152.364
C08987=1097.177,289.255,419.999,178.180,18.639,152.364
C08988=1097.186,289.627,419.955,178.185,18.642,152.364
C08989=1097.195,289.999,419.911,178.190,18.646,152.364
C08990=1097.203,290.369,419.866,178.194,18.648,152.363
C08991=1097.208,290.618,419.837,178.198,18.650,152.363
C08992=1097.214,290.866,419.807,178.201,18.652,152.363
C08993=1097.220,291.114,419.777,178.204,18.655,152.363
C08994=1097.226,291.362,419.747,178.208,18.657,152.363
C08995=1097.232,291.610,419.717,178.211,18.659,152.363
C08996=1097.237,291.858,419.688,178.214,18.661,152.363
C08997=1097.243,292.107,419.658,178.218,18.663,152.363
C08998=1097.249,292.355,419.628,178.221,18.666,152.363
C08999=1097.254,292.603,419.598,178.224,18.668,152.362
C09000=1097.260,292.851,419.568,178.228,18.670,152.362
C09001=1097.265,293.099,419.538,178.231,18.672,152.362
C09002=1097.271,293.347,419.508,178.234,18.674,152.362
C09003=1097.277,293.596,419.478,178.237,18.676,152.362
C09004=1097.283,293.843,419.448,178.240,18.678,152.362
C09005=1097.288,294.092,419.418,178.244,18.680,152.362
C09006=1097.294,294.340,419.388,178.247,18.682,152.362
C09007=1097.299,294.588,419.358,178.250,18.685,152.362
C09008=1097.305,294.835,419.328,178.253,18.687,152.361
C09009=1097.311,295.084,419.297,178.257,18.689,152.361
C09010=1097.317,295.332,419.268,178.260,18.691,152.361
C09011=1097.322,295.580,419.237,178.263,18.693,152.361
C09012=1097.328,295.829,419.208,178.267,18.696,152.361
C09013=1097.334,296.076,419.177,178.270,18.698,152.361
C09014=1097.340,296.324,419.147,178.273,18.700,152.361
C09015=1097.345,296.573,419.117,178.277,18.702,152.361
C09016=1097.351,296.820,419.087,178.280,18.704,152.361
C09017=1097.357,297.068,419.057,178.283,18.707,152.361
C09018=1097.361,297.317,419.026,178.286,18.709,152.360
C09019=1097.367,297.565,418.996,178.290,18.711,152.360
C09020=1097.373,297.813,418.966,178.293,18.713,152.360
C09021=1097.379,298.060,418.935,178.296,18.716,152.360
C09022=1097.384,298.309,418.906,178.300,18.718,152.360
C09023=1097.390,298.557,418.875,178.303,18.720,152.360
C09024=1097.395,298.805,418.844,178.306,18.722,152.360
C09025=1097.401,299.053,418.814,178.309,18.725,152.360
C09026=1097.407,299.301,418.784,178.313,18.727,152.360
C09027=1097.412,299.549,418.753,178.316,18.729,152.360
C09028=1097.418,299.797,418.723,178.319,18.732,152.360
C09029=1097.423,300.045,418.693,178.322,18.734,152.360
C09030=1097.428,300.293,418.662,178.326,18.736,152.360
C09031=1097.434,300.541,418.631,178.329,18.738,152.360
C09032=1097.440,300.789,418.601,178.332,18.741,152.359
C09033=1097.445,301.037,418.570,178.335,18.743,152.359
C09034=1097.451,301.285,418.540,178.338,18.746,152.359
C09035=1097.456,301.533,418.509,178.342,18.748,152.359
C09036=1097.462,301.781,418.478,178.345,18.750,152.359
C09037=1097.468,302.029,418.448,178.348,18.753,152.359
C09038=1097.473,302.277,418.417,178.351,18.755,152.359
C09039=1097.483,302.662,418.369,178.356,18.758,152.359
C09040=1097.490,303.047,418.322,178.361,18.762,152.359
C09041=1097.500,303.432,418.275,178.366,18.766,152.359
C09042=1097.508,303.818,418.227,178.372,18.770,152.359
C09043=1097.514,304.066,418.196,178.375,18.772,152.359
C09044=1097.519,304.314,418.165,178.378,18.774,152.359
C09045=1097.525,304.562,418.135,178.381,18.776,152.359
C09046=1097.531,304.810,418.103,178.384,18.779,152.359
C09047=1097.536,305.058,418.073,178.388,18.781,152.359
C09048=1097.542,305.306,418.042,178.391,18.784,152.359
C09049=1097.547,305.554,418.011,178.394,18.786,152.359
C09050=1097.554,305.802,417.981,178.397,18.788,152.359
C09051=1097.559,306.050,417.949,178.401,18.791,152.359
C09052=1097.565,306.297,417.919,178.404,18.793,152.359
C09053=1097.570,306.546,417.888,178.407,18.795,152.358
C09054=1097.576,306.793,417.857,178.410,18.798,152.358
C09055=1097.582,307.042,417.825,178.414,18.800,152.358
C09056=1097.588,307.289,417.795,178.417,18.803,152.358
C09057=1097.593,307.538,417.764,178.420,18.805,152.358
C09058=1097.599,307.785,417.734,178.423,18.807,152.358
C09059=1097.605,308.034,417.702,178.426,18.810,152.358
C09060=1097.610,308.281,417.671,178.430,18.813,152.358
C09061=1097.616,308.529,417.640,178.433,18.815,152.358
C09062=1097.621,308.778,417.608,178.437,18.817,152.358
C09063=1097.627,309.026,417.578,178.440,18.820,152.358
C09064=1097.633,309.273,417.546,178.443,18.822,152.358
C09065=1097.639,309.522,417.516,178.446,18.825,152.358
C09066=1097.644,309.769,417.484,178.450,18.827,152.358
C09067=1097.650,310.017,417.454,178.453,18.830,152.358
C09068=1097.656,310.265,417.421,178.456,18.832,152.358
C09069=1097.661,310.513,417.391,178.459,18.834,152.358
C09070=1097.667,310.761,417.360,178.462,18.837,152.358
C09071=1097.673,311.009,417.328,178.465,18.839,152.358
C09072=1097.679,311.257,417.297,178.469,18.842,152.358
C09073=1097.684,311.505,417.266,178.472,18.844,152.358
C09074=1097.690,311.753,417.234,178.476,18.847,152.358
C09075=1097.696,312.001,417.204,178.479,18.849,152.358
C09076=1097.702,312.249,417.172,178.482,18.852,152.358
C09077=1097.707,312.497,417.141,178.485,18.854,152.358
C09078=1097.713,312.744,417.110,178.489,18.857,152.358
C09079=1097.719,312.993,417.078,178.492,18.859,152.358
C09080=1097.724,313.241,417.047,178.495,18.862,152.358
C09081=1097.731,313.489,417.015,178.498,18.864,152.358
C09082=1097.737,313.736,416.984,178.501,18.867,152.358
C09083=1097.742,313.985,416.952,178.504,18.869,152.358
C09084=1097.748,314.232,416.921,178.507,18.872,152.358
C09085=1097.754,314.480,416.889,178.511,18.875,152.358
C09086=1097.759,314.728,416.858,178.515,18.877,152.358
C09087=1097.766,314.976,416.827,178.518,18.880,152.358
C09088=1097.771,315.224,416.795,178.521,18.882,152.358
C09089=1097.777,315.472,416.763,178.524,18.885,152.358
C09090=1097.783,315.720,416.732,178.527,18.887,152.358
C09091=1097.791,316.108,416.682,178.532,18.892,152.358
C09092=1097.800,316.496,416.633,178.537,18.896,152.358
C09093=1097.808,316.883,416.583,178.542,18.899,152.358
C09094=1097.817,317.270,416.534,178.547,18.904,152.358
C09095=1097.823,317.519,416.502,178.550,18.907,152.358
C09096=1097.828,317.767,416.471,178.553,18.909,152.358
C09097=1097.834,318.015,416.439,178.556,18.912,152.358
C09098=1097.840,318.263,416.407,178.560,18.915,152.358
C09099=1097.846,318.511,416.375,178.563,18.918,152.358
C09100=1097.851,318.758,416.343,178.566,18.920,152.359
